# B&R Automation Studio project GAT
Automation Studio 4.10.3.60 SP; technology packages: mapp 5.16.1, mappCockpit 5.16.0, mappControl 5.16.0, mappMotion 5.16.0, mappView 5.16.1

## Configuration 4PPC50_101E_10B

CPU 4PPC50.101E-10B, AutomationRuntime C4.91, Build 4.1.2, Safety 0.0, Vc 

### Task classes (Cpu.sw)
```
Cyclic#1 (cycle 1600 us, tolerance 1600 us):
  MainCtrl <- MainControl.MainCtrl.prg [disabled]
  CrossCutte <- MachineControl.CrossCutter.CrossCutter.prg
  Conveyor <- MachineControl.Conveyor.Conveyor.prg
  AlarmUI <- (binary)
Cyclic#2 (cycle 20000 us, tolerance 20000 us):
  AlarmMgt <- Infrastructure.Alarm.AlarmMgt.prg
Cyclic#4 (cycle 80000 us, tolerance 80000 us):
  AuditMgt <- Infrastructure.Audit.AuditMgt.prg
  ReportMgt <- Infrastructure.Report.ReportMgt.prg
  DataMgt <- Infrastructure.Data.DataMgt.prg
  ProcessCon <- Infrastructure.SysServices.ProcessConfig.prg [disabled]
  PIDControl <- MainControl.PIDControl.prg [disabled]
  RecipeMgt <- Infrastructure.Recipe.RecipeMgt.prg
  IoBrowser <- Infrastructure.SysServices.IoBrowser.prg
  UsbDevLink <- Infrastructure.UsbDevLink.UsbDevLink.prg
Cyclic#5 (cycle 200000 us, tolerance 200000 us):
  SysServs <- Infrastructure.SysServices.SysServs.prg
Cyclic#8 (cycle 8000 us, tolerance 30000000 us):
  UserXMgt <- Infrastructure.UserX.UserXMgt.prg
  UserMgt <- Infrastructure.User.UserMgt.prg [disabled]
DataObjects: McAcpSys
NcDataObjects: McDriveLog
Binaries: arsvcreg, FWRules, McAcpDrv, McAcpSim, mvLoader, McProfGen, McMechSys, TCData, TCLang, udbdef, arcoal, arflatprv, mCoWebSc, OpcUaSrv, arconfig, User, Role, iomap, asfw, ashwac, ashwd, sysconf, TC, Report, Rcp, AlmHistory, Data, Audit, UserXlogin, UsX, Settings, AxCfg, Alarm, CutCamAut, myUnits, FileMgr, CutterAlm, ConvGrp, MachineGrp, Cutter, ConvAlm, CutterGrp, aruser, File, FileMgrRep, FileMgrDat, FileMgrAud, FileUI, CamAutoMa1, User_1, Config, Config_32, AlmCutter, Config_1, Config_2, UserMgr, UserSign, UserLogin, profiler, Config_31, Config_3, CfgUser, Login, Config_23, Config_24, Config_21, Config_20, CamAutoMat, vConfig_0, Config_0, Config_13, Config_5, Config_8, Config_9, Config_11, Config_15, Config_14, Config_12, Config_10, Config_6, Config_7, Config_22, Config_4, Master, Slave, CamID, CamList, ProfGen, vMaster
Libraries: McBase, McAcpAx, McPathGen, McPureVAx, McAxGroup, McAxis, McAcpPar, McProgInt, MpTool, MpAxis, MpBase, MpWebXs, MpAudit, MpRecipe, MpReport, MpFile, MpAlarmX, MpCom, MpBackup, AsArSdm, FileIO, astime, sys_lib, runtime, MpServer, MpData, DataObj, brsystem, CoTrace, AsZip, MpUserX, AsUPS, MTBasics, MTTypes, Gat, AsIO, AsBrStr, AsIOMMan, IoMapMan, ArCfgMan, AsUSB, powerlnk, arssl, arproject, asarlog, asarprof, asmem, asarcfg, asieccon, asstring, asepl, aseth, ashw, arcert, dvframe, standard, mpregmark
```

### Hardware
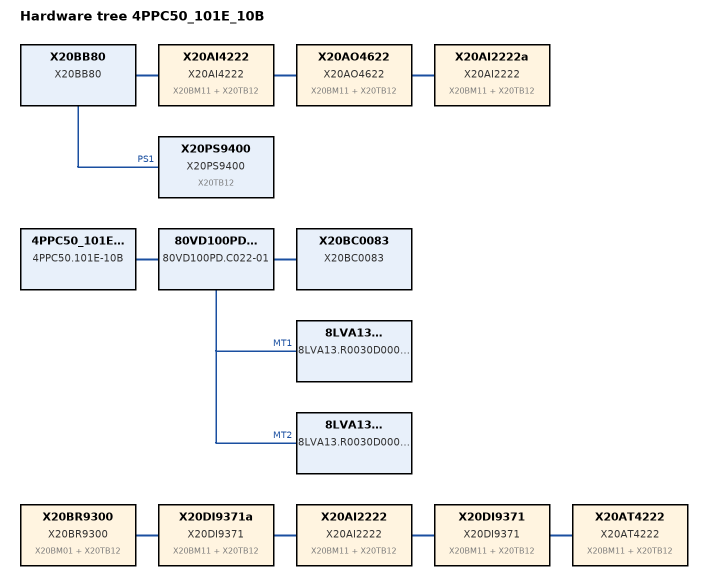
```
4PPC50_101E_10B : 4PPC50.101E-10B v1.1.2.1
  Connector IF1:
    CycleTime = 800
  Connector IF2:
    ActivateDevice = 1
    Mode = Manual
    InternetAddress = 10.86.50.12
    SubnetMask = 255.255.255.0
  Connector IF3:
    AssignedOperatingSystem = ARemb
  Connector IF4:
    AssignedOperatingSystem = GPOS
  ConfigurationID = GAT_10inC50_4PPC50_101E_10B
  UserPartitionSize = 25
  UserRamSize = 16000
  RemMemSize = 48000
  TimerDeviceType = EPLX2X
  TimerDevice = 4PPC50_101E_10B.IF1
  TaskClassIdleTime = 4000
  Cyclic1Duration = 1600
  Cyclic1Tolerance = 1600
  Cyclic1Stack = 16384
  Cyclic2Duration = 20000
  Cyclic2Tolerance = 20000
  Cyclic3Duration = 40000
  Cyclic3Tolerance = 40000
  Cyclic4Duration = 80000
  Cyclic4Tolerance = 80000
  Cyclic4Stack = 16384
  Cyclic5Duration = 200000
  Cyclic5Tolerance = 200000
  Cyclic6Duration = 500000
  Cyclic6Tolerance = 500000
  Cyclic7Duration = 1000000
  Cyclic7Tolerance = 1000000
  Cyclic8Duration = 8000
  Cyclic8Tolerance = 30000000
  FileDevice1
  FileDeviceName1 = mappRecipe
  FileDevicePath1 = F:\GAT\Recipe
  FileDevice2
  FileDeviceName2 = mappAudit
  FileDevicePath2 = F:\GAT\Audit
  FileDevice3
  FileDeviceName3 = mappReport
  FileDevicePath3 = F:\GAT\Report
  FileDevice4
  FileDeviceName4 = mappData
  FileDevicePath4 = F:\GAT\Data
  TimeZone = 295
  EthernetDefaultGateway = 10.86.13.1
  FTPProtocol = 2
  FtpUser1
  FtpUsername1 = BR
  FtpUserPassword1 = GhNaeKiLvl7cP7K0k5JDdXf+fyc8NJfckbGpEUwY4Hg=  // FTP
  FtpUserSalt1 = zT8zXD9V
  FTPAccessRight1 = 0
  FTPdevice1 = ALL
  ActivateOpcUa = 1
  OpcUaActivateAuditEvents = 1
  OpcUa_Security_AdminRole = Administrators
  OpcUaInformationModels_PV_Version = 1
  LXTMode = Manual
  LXTInternetAddress = 10.86.50.13
  LXTSubnetmask = 255.255.255.0
80VD100PD.C022-01 : 80VD100PD.C022-01 v2.5.0.0  [PLK1 -> 4PPC50_101E_10B.IF1 (NodeNumber=1) [Cable Type=PowerlinkCable, Length=10, Version=1.0.0.3]; PLK2 -> X20BC0083.PLK1 (NodeNumber=1) [Cable Type=PowerlinkCable, Length=10, Version=1.0.0.3]; MT2 -> 8LVA13.R0030D000-0a.MT]
  DriveConfiguration/Module:
    McAcoposTypeID = AcoposMicroDConfig
    ActivateACOPOSSimulationOnPLC = 1
  DriveConfiguration/Encoder/EncoderX6A/InterfaceType:
    ResolverPolepairs = 1
  DriveConfiguration/Encoder/EncoderX6B/InterfaceType:
    ResolverPolepairs = 1
  DriveConfiguration/Channel[1]/RealAxis:
    AxisReference = gAxisConveyor
  DriveConfiguration/Channel[1]/RealAxis/MechanicalElements/Gearbox:
    InputIsReadOnly = 0
    Input = 1
    OutputIsReadOnly = 0
    Output = 1
  DriveConfiguration/Channel[1]/RealAxis/MechanicalElements/RotaryToLinearTransformation:
    ReferenceDistanceIsReadOnly = 0
    ReferenceDistance = 1
  DriveConfiguration/Channel[1]/RealAxis/Controller:
    ModeIsReadOnly = 0
    Mode = PositionController
  DriveConfiguration/Channel[1]/RealAxis/Controller/Mode/Position:
    ProportionalGain = 50.0
    IntegrationTime = 0.0
    PredictionTime = 0.0004
    TotalDelayTime = 0.0004
  DriveConfiguration/Channel[1]/RealAxis/Controller/Mode/Speed:
    ProportionalGainIsReadOnly = 0
    ProportionalGain = 2.0
    IntegrationTimeIsReadOnly = 0
    IntegrationTime = 0.0
    FilterTimeIsReadOnly = 0
    FilterTime = 0.0
  DriveConfiguration/Channel[1]/RealAxis/Controller/Mode/LoopFilters:
    LoopFilter1 = NotUsed
    LoopFilter2 = NotUsed
    LoopFilter3 = NotUsed
  DriveConfiguration/Channel[1]/RealAxis/Homing:
    Mode = Direct
  DriveConfiguration/Channel[1]/RealAxis/Homing/Mode:
    Position = 0.0
    ReferencePulse = NotUsed
  DriveConfiguration/Channel[1]/RealAxis/Homing:
    RestorePositionVariable = 
  DriveConfiguration/Channel[1]/RealAxis/StopReaction:
    Quickstop = DecelerationLimit
    DriveError = DecelerationLimit
  DriveConfiguration/Channel[1]/RealAxis/MovementErrorLimits:
    PositionError = 1.0
    VelocityErrorMonitoring = Automatic1
  DriveConfiguration/Channel[1]/RealAxis:
    JerkFilter = NotUsed
  DriveConfiguration/Channel[1]/RealAxis/DigitalInputs/HomingSwitch:
    Source = NotUsed
    Level = High
  DriveConfiguration/Channel[1]/RealAxis/DigitalInputs/PositiveLimitSwitch:
    Source = NotUsed
    Level = High
  DriveConfiguration/Channel[1]/RealAxis/DigitalInputs/NegativeLimitSwitch:
    Source = NotUsed
    Level = High
  DriveConfiguration/Channel[1]/RealAxis/DigitalInputs/Trigger1:
    Source = X2Trigger1
    Level = High
  DriveConfiguration/Channel[1]/RealAxis/DigitalInputs/Trigger2:
    Source = X2Trigger2
    Level = High
  DriveConfiguration/Channel[1]/RealAxis/DigitalInputs/Quickstop:
    Input = Trigger2
  DriveConfiguration/Channel[1]/RealAxis/Simulation:
    SimulationModeOnPLC = SetValueGeneration
    SimulationModeOnACOPOS = NotUsed
  DriveConfiguration/Channel[2]/RealAxis:
    AxisReference = gAxisCrossCutter
  DriveConfiguration/Channel[2]/RealAxis/MechanicalElements/Gearbox:
    InputIsReadOnly = 0
    Input = 1
    OutputIsReadOnly = 0
    Output = 1
  DriveConfiguration/Channel[2]/RealAxis/MechanicalElements/RotaryToLinearTransformation:
    ReferenceDistanceIsReadOnly = 0
    ReferenceDistance = 1
  DriveConfiguration/Channel[2]/RealAxis/Controller:
    ModeIsReadOnly = 0
    Mode = PositionController
  DriveConfiguration/Channel[2]/RealAxis/Controller/Mode/Position:
    ProportionalGain = 50.0
    IntegrationTime = 0.0
    PredictionTime = 0.0004
    TotalDelayTime = 0.0004
  DriveConfiguration/Channel[2]/RealAxis/Controller/Mode/Speed:
    ProportionalGainIsReadOnly = 0
    ProportionalGain = 2.0
    IntegrationTimeIsReadOnly = 0
    IntegrationTime = 0.0
    FilterTimeIsReadOnly = 0
    FilterTime = 0.0
  DriveConfiguration/Channel[2]/RealAxis/Controller/Mode/LoopFilters:
    LoopFilter1 = NotUsed
    LoopFilter2 = NotUsed
    LoopFilter3 = NotUsed
  DriveConfiguration/Channel[2]/RealAxis/Homing:
    Mode = Direct
  DriveConfiguration/Channel[2]/RealAxis/Homing/Mode:
    Position = 0.0
    ReferencePulse = NotUsed
  DriveConfiguration/Channel[2]/RealAxis/Homing:
    RestorePositionVariable = 
  DriveConfiguration/Channel[2]/RealAxis/StopReaction:
    Quickstop = DecelerationLimit
    DriveError = DecelerationLimit
  DriveConfiguration/Channel[2]/RealAxis/MovementErrorLimits:
    PositionError = 1.0
    VelocityErrorMonitoring = Automatic1
  DriveConfiguration/Channel[2]/RealAxis:
    JerkFilter = NotUsed
  DriveConfiguration/Channel[2]/RealAxis/DigitalInputs/HomingSwitch:
    Source = NotUsed
    Level = High
  DriveConfiguration/Channel[2]/RealAxis/DigitalInputs/PositiveLimitSwitch:
    Source = NotUsed
    Level = High
  DriveConfiguration/Channel[2]/RealAxis/DigitalInputs/NegativeLimitSwitch:
    Source = NotUsed
    Level = High
  DriveConfiguration/Channel[2]/RealAxis/DigitalInputs/Trigger1:
    Source = X2Trigger1
    Level = High
  DriveConfiguration/Channel[2]/RealAxis/DigitalInputs/Trigger2:
    Source = X2Trigger2
    Level = High
  DriveConfiguration/Channel[2]/RealAxis/DigitalInputs/Quickstop:
    Input = Trigger2
  DriveConfiguration/Channel[2]/RealAxis/Simulation:
    SimulationModeOnPLC = SetValueGeneration
    SimulationModeOnACOPOS = NotUsed
  DriveConfiguration/Channel[2]/RealAxis/AxisFeatures:
    FeatureRef[1] = CutterCamAutomat
8LVA13.R0030D000-0 : 8LVA13.R0030D000-0 v2.2.0.4  [MT -> 80VD100PD.C022-01.MT1]
  M1/MotorParameters:
    MOTOR_AMB_TEMP_RATED = 40
8LVA13.R0030D000-0a : 8LVA13.R0030D000-0 v2.2.0.4  [MT -> 80VD100PD.C022-01.MT2]
  M1/MotorParameters:
    MOTOR_AMB_TEMP_RATED = 40
X20AI2222 : X20AI2222 v1.1.0.0  [SS1 -> X20TB12b.SS; SL -> X20BM11a.SL1]
  Supervision = off
X20AI2222a : X20AI2222 v1.1.0.0  [SS1 -> X20TB12h.SS; SL -> X20BM11f.SL1]
  Supervision = off
X20AI4222 : X20AI4222 v1.1.0.0  [SS1 -> X20TB12f.SS; SL -> X20BM11d.SL1]
X20AO4622 : X20AO4622 v1.2.0.0  [SS1 -> X20TB12g.SS; SL -> X20BM11e.SL1]
X20AT4222 : X20AT4222 v1.3.0.0  [SS1 -> X20TB12a.SS; SL -> X20BM11.SL1]
  Supervision = off
X20BB80 : X20BB80 v1.0.2.0
X20BC0083 : X20BC0083 v2.11.1.0  [PLK1 -> 80VD100PD.C022-01.PLK2 (NodeNumber=2) [Cable Type=PowerlinkCable, Length=10, Version=1.0.0.3]; SL -> X20BB80.SL1]
X20BM01 : X20BM01 v2.1.0.0
X20BM11 : X20BM11 v1.0.0.1  [X2X1 -> X20BM11b.X2X2]
X20BM11a : X20BM11 v1.0.0.1  [X2X1 -> X20BM11c.X2X2]
X20BM11b : X20BM11 v1.0.0.1  [X2X1 -> X20BM11a.X2X2]
X20BM11c : X20BM11 v1.0.0.1  [X2X1 -> X20BM01.X2X2]
X20BM11d : X20BM11 v1.0.0.1  [X2X1 -> X20BB80.IF1]
X20BM11e : X20BM11 v1.0.0.1  [X2X1 -> X20BM11d.X2X2]
X20BM11f : X20BM11 v1.0.0.1  [X2X1 -> X20BM11e.X2X2]
X20BR9300 : X20BR9300 v1.1.0.0  [SS1 -> X20TB12.SS; SL -> X20BM01.SL1; X2X1 -> 4PPC50_101E_10B.IF5 [Cable Type=X2XCable, Length=10, Version=1.0.0.3]]
  Supervision = off
X20DI9371 : X20DI9371 v1.1.0.0  [SS1 -> X20TB12c.SS; SL -> X20BM11b.SL1]
X20DI9371a : X20DI9371 v1.1.0.0  [SS1 -> X20TB12d.SS; SL -> X20BM11c.SL1]
X20PS9400 : X20PS9400 v1.5.0.0  [SS1 -> X20TB12e.SS; PS -> X20BB80.PS1]
X20TB12 : X20TB12 v1.0.0.0
X20TB12a : X20TB12 v1.0.0.0
X20TB12b : X20TB12 v1.0.0.0
X20TB12c : X20TB12 v1.0.0.0
X20TB12d : X20TB12 v1.0.0.0
X20TB12e : X20TB12 v1.0.0.0
X20TB12f : X20TB12 v1.0.0.0
X20TB12g : X20TB12 v1.0.0.0
X20TB12h : X20TB12 v1.0.0.0
```

### IoMap.iom - 4PPC50_101E_10B/IoMap.iom
```iecst
VAR_CONFIG
	::SysServs:CpuIoMap.SerialNumber_CPU AT %ID."4PPC50_101E_10B".SerialNumber_CPU;
	::SysServs:CpuIoMap.ModuleID_CPU AT %IW."4PPC50_101E_10B".ModuleID_CPU;
	::SysServs:CpuIoMap.HardwareVariant AT %IW."4PPC50_101E_10B".HardwareVariant;
	::SysServs:CpuIoMap.FirmwareVersion AT %IW."4PPC50_101E_10B".FirmwareVersion;
	::SysServs:CpuIoMap.TemperatureCPU AT %IW."4PPC50_101E_10B".TemperatureCPU;
	::SysServs:CpuIoMap.TemperatureENV AT %IW."4PPC50_101E_10B".TemperatureENV;
	::SysServs:CpuIoMap.TerminalTemperatureCPU AT %IW."4PPC50_101E_10B".TerminalTemperatureCPU;
	::SysServs:CpuIoMap.TerminalOK AT %IX."4PPC50_101E_10B".TerminalOk;
	::SysServs:CpuIoMap.TerminalStatus AT %IB."4PPC50_101E_10B".TerminalStatus;
	::SysServs:CpuIoMap.TerminalLoadCPU0 AT %IB."4PPC50_101E_10B".TerminalLoadCPU0;
	::SysServs:CpuIoMap.TerminalLoadCPU1 AT %IB."4PPC50_101E_10B".TerminalLoadCPU1;
	::AlarmMgt:SafetyInputs.SafetyPLC AT %IX."X20DI9371".DigitalInput02;
	::AlarmMgt:SafetyInputs.EmergencyStop[0]  AT %IX."X20DI9371a".DigitalInput06;
END_VAR
```

### AxCfg.axis - 4PPC50_101E_10B/mappMotion/AxCfg.axis
```
Element gAxisConveyor (Type=axis)
  BaseTypeIsReadOnly = 0
  BaseType = Linear
    MeasurementUnit = 5066068
    MeasurementResolutionIsReadOnly = 0
    MeasurementResolution = 0.01
    CountDirectionIsReadOnly = 0
    CountDirection = Standard
  MovementLimitsIsReadOnly = 0
  MovementLimits = Internal
    Position:
      LowerLimitMin = -1.79769313486231E308
      UpperLimitMax = 1.79769313486231E308
      LowerLimit = -1000000000000000000000.0
      UpperLimit = 1000000000000000000000.0
    VelocityIsReadOnly = 0
    Velocity:
      VelocityMax = 3.4E38
      Velocity = 10000
    AccelerationIsReadOnly = 0
    Acceleration:
      AccelerationMax = 3.4E38
      Acceleration = 50000
    DecelerationIsReadOnly = 0
    Deceleration:
      DecelerationMax = 3.4E38
      Deceleration = 50000
  Alarms = MpAlarmX
    mapp.AlarmX.Core.Configuration:
      [0]:
        Message = {$MpMotion/Alarms/System}
      [1]:
        Message = {$MpMotion/Alarms/Initialization}
      [2]:
        Message = {$MpMotion/Alarms/Parameter}
      [3]:
        Message = {$MpMotion/Alarms/Operation}
      [4]:
        Message = {$MpMotion/Alarms/DataAccess}
      [5]:
        Message = {$MpMotion/Alarms/Syntax}
      [9]:
        Message = {$MpMotion/Alarms/Network}
      [10]:
        Message = {$MpMotion/Alarms/Encoder}
        AdditionalInformation1 = Something wrong with the encoder inside the motor
      [11]:
        Message = {$MpMotion/Alarms/Drive}
        AdditionalInformation1 = Acopos Drive Error
      [12]:
        Message = {$MpMotion/Alarms/IO}
      [13]:
        Message = {$MpMotion/Alarms/Supply}
      [14]:
        Message = {$MpMotion/Alarms/Motor}
      [15]:
        Message = {$MpMotion/Alarms/HoldingBrake}
Element gAxisCrossCutter (Type=axis)
  BaseTypeIsReadOnly = 0
  BaseType = RotaryPeriodic
    MeasurementUnitIsReadOnly = 0
    MeasurementUnit = 17476
    MeasurementResolutionIsReadOnly = 0
    MeasurementResolution = 0.01
    CountDirectionIsReadOnly = 0
    CountDirection = Inverse
    PeriodSettings:
      Period = 360
  MovementLimitsIsReadOnly = 0
  MovementLimits = Internal
    Position:
      LowerLimitMin = -1.79769313486231E308
      UpperLimitMax = 1.79769313486231E308
      LowerLimit = -1000.0
      UpperLimit = 1000.0
    VelocityIsReadOnly = 0
    Velocity:
      VelocityMax = 3.4E38
      Velocity = 500000
    AccelerationIsReadOnly = 0
    Acceleration:
      AccelerationMax = 3.4E38
      Acceleration = 5000000
    DecelerationIsReadOnly = 0
    Deceleration:
      DecelerationMax = 3.4E38
      Deceleration = 5000000
  Alarms = MpAlarmX
    mapp.AlarmX.Core.Configuration:
      [0]:
        Message = {$MpMotion/Alarms/System}
      [1]:
        Message = {$MpMotion/Alarms/Initialization}
      [2]:
        Message = {$MpMotion/Alarms/Parameter}
      [3]:
        Message = {$MpMotion/Alarms/Operation}
      [4]:
        Message = {$MpMotion/Alarms/DataAccess}
      [5]:
        Message = {$MpMotion/Alarms/Syntax}
      [9]:
        Message = {$MpMotion/Alarms/Network}
      [10]:
        Message = {$MpMotion/Alarms/Encoder}
      [11]:
        Message = {$MpMotion/Alarms/Drive}
      [12]:
        Message = {$MpMotion/Alarms/IO}
      [13]:
        Message = {$MpMotion/Alarms/Supply}
      [14]:
        Message = {$MpMotion/Alarms/Motor}
      [15]:
        Message = {$MpMotion/Alarms/HoldingBrake}
```

### Alarm.mpalarmxcore - 4PPC50_101E_10B/mappServices/Alarm.mpalarmxcore
```
Element gAlarmXMpLink (Type=mpalarmxcore)
  mapp.AlarmX.Core:
    Mapping:
      [0]:
        Alarm = gAxisMaster*
        [0] = Reaction
          Name = MasterWaitAcknowledge
      [1]:
        Alarm = gAxisSlave*
        [0] = Reaction
          Name = SlaveWaitAcknowledge
    BySeverity:
      [0]:
        Severity = 1
        [0] = Reaction
          Name = StopMovements
      [1]:
        Severity = 10
        [0] = Reaction
      [2]:
        Severity = 20
        [0] = Reaction
  mapp.AlarmX.Core.Configuration:
    [0]:
      Name = FeederSpeedNotSet
      Message = {$AlarmTexts/FeederSpeedNotSet}
      Code = 250
      Severity = 10
    [1]:
      Name = CutterSpeedNotSet
      Message = {$AlarmTexts/CutterSpeedNotSet}
      Code = 251
      Severity = 10
    [2]:
      Name = CutterPositionNotSet
      Message = {$AlarmTexts/CutterPositionNotSet}
      Code = 252
      Severity = 10
    [3]:
      Name = PidOscTuningError
      Message = {$AlarmTexts/PidOscTuningError}
      Behavior = DiscreteValueMonitoring
        Monitoring:
          MonitoredPV = ::PIDControl:MTBasicsOscillationTuning_0.StatusID
          TriggerValues:
            [0] = -1999999999..-1000000000
    [4]:
      Name = PidControlError
      Message = {$AlarmTexts/PidControlError}
      Behavior = DiscreteValueMonitoring
        Monitoring:
          MonitoredPV = ::PIDControl:MTBasicsPID_0.StatusID
          TriggerValues:
            [0] = -1999999999..-1000000000
    [5]:
      Name = PidControlWarning
      Message = {$AlarmTexts/PidControlWarning}
      Behavior = DiscreteValueMonitoring
        Monitoring:
          MonitoredPV = ::PIDControl:MTBasicsPID_0.StatusID
          TriggerValues:
            [0] = -2999999999..-2000000000
    [6]:
      Name = SetCamFailed
      Message = {$AlarmTexts/SetCamFailed}
    [7]:
      Name = EmergencyStop_0
      Message = {$AlarmTexts/EmergencyStop.0}
      Behavior = DiscreteValueMonitoring
        Recording:
          ActiveToInactive = TRUE
        Monitoring:
          MonitoredPV = ::AlarmMgt:SafetyInputs.EmergencyStop[0]
          TriggerValues:
            [0] = 1
    [8]:
      Name = EmergencyStop_1
      Message = {$AlarmTexts/EmergencyStop.1}
      Behavior = DiscreteValueMonitoring
        Recording:
          ActiveToInactive = TRUE
        Monitoring:
          MonitoredPV = ::AlarmMgt:SafetyInputs.EmergencyStop[1]
          TriggerValues:
            [0] = 1
    [9]:
      Name = EmergencyStop_2
      Message = {$AlarmTexts/EmergencyStop.2}
      Behavior = DiscreteValueMonitoring
        Recording:
          ActiveToInactive = TRUE
        Monitoring:
          MonitoredPV = ::AlarmMgt:SafetyInputs.EmergencyStop[2]
          TriggerValues:
            [0] = 1
    [10]:
      Name = SafetyDoor_0
      Message = {$AlarmTexts/SafetyDoor.0}
      Behavior = DiscreteValueMonitoring
        Recording:
          ActiveToInactive = TRUE
        Monitoring:
          MonitoredPV = ::AlarmMgt:SafetyInputs.SafetyDoor[0]
          TriggerValues:
            [0] = 1
    [11]:
      Name = SafetyDoor_1
      Message = {$AlarmTexts/SafetyDoor.1}
      Behavior = DiscreteValueMonitoring
        Recording:
          ActiveToInactive = TRUE
        Monitoring:
          MonitoredPV = ::AlarmMgt:SafetyInputs.SafetyDoor[1]
          TriggerValues:
            [0] = 1
    [12]:
      Name = SafetyDoor_2
      Message = {$AlarmTexts/SafetyDoor.2}
      Behavior = DiscreteValueMonitoring
        Recording:
          ActiveToInactive = TRUE
        Monitoring:
          MonitoredPV = ::AlarmMgt:SafetyInputs.SafetyDoor[2]
          TriggerValues:
            [0] = 1
    [13]:
      Name = SafetyDoor_3
      Message = {$AlarmTexts/SafetyDoor.3}
      Behavior = DiscreteValueMonitoring
        Recording:
          ActiveToInactive = TRUE
        Monitoring:
          MonitoredPV = ::AlarmMgt:SafetyInputs.SafetyDoor[3]
          TriggerValues:
            [0] = 1
    [14]:
      Name = SafetyDoor_4
      Message = {$AlarmTexts/SafetyDoor.4}
      Behavior = DiscreteValueMonitoring
        Recording:
          ActiveToInactive = TRUE
        Monitoring:
          MonitoredPV = ::AlarmMgt:SafetyInputs.SafetyDoor[4]
          TriggerValues:
            [0] = 1
    [15]:
      Name = SafetyDoor_5
      Message = {$AlarmTexts/SafetyDoor.5}
      Behavior = DiscreteValueMonitoring
        Recording:
          ActiveToInactive = TRUE
        Monitoring:
          MonitoredPV = ::AlarmMgt:SafetyInputs.SafetyDoor[5]
          TriggerValues:
            [0] = 1
    [16]:
      Name = SafetyPLC
      Message = {$AlarmTexts/SafetyPLC}
      Behavior = DiscreteValueMonitoring
        Recording:
          ActiveToInactive = TRUE
        Monitoring:
          MonitoredPV = ::AlarmMgt:SafetyInputs.SafetyPLC
          TriggerValues:
            [0] = 1
  mapp.AlarmX.Core.Snippets:
    AutoDetect = 1
    [0]:
      Key = CutterSpeed
      Value:
        PV = ::MainCtrl:AxisControl[1].Status.ActVelocity
    [1]:
      Key = CutterPosition
      Value:
        PV = ::MainCtrl:AxisControl[1].Status.ActPosition
    [2]:
      Key = PidTuningError
      Value:
        PV = ::PIDControl:MTBasicsOscillationTuning_0.StatusID
    [3]:
      Key = PidControlError
      Value:
        PV = ::PIDControl:MTBasicsPID_0.StatusID
  mapp.AlarmX.Core.Categories:
    [0]:
      Name = Information
      SourceProperty:
        Severity = 20
    [1]:
      Name = Warning
      SourceProperty:
        Severity = 10
    [2]:
      Name = Error
      SourceProperty:
        Severity = 1
```

### AlmHistory.mpalarmxhistory - 4PPC50_101E_10B/mappServices/AlmHistory.mpalarmxhistory
```
Element gAlarmXHistoryMpLink (Type=mpalarmxhistory)
  mapp.AlarmX.History:
    Memory:
      MemorySize = 6000
    Auditing = MpAudit
```

### ConvAlm.mpalarmxcore - 4PPC50_101E_10B/mappServices/Conveyor/ConvAlm.mpalarmxcore
```
Element gAlarmXCore_Conveyor (Type=mpalarmxcore)
  mapp.AlarmX.Core:
    BySeverity:
      [0]:
        Severity = 1..9
        [0] = Reaction
          Name = Info
        [1] = Escalate
      [1]:
        Severity = 10..19
        [0] = Reaction
          Name = Warning
        [1] = Escalate
      [2]:
        Severity = 20..29
        [0] = Reaction
          Name = Alarm
        [1] = Escalate
      [3]:
        Severity = 30..39
        [0] = Reaction
          Name = Safety
        [1] = Escalate
  mapp.AlarmX.Core.Configuration:
    [0]:
      Name = ReferenceRequired
      Message = {$IAT/Conveyor/Info/Name} : {$IAT/Conveyor/Alarms/ReferenceRequired}
      Severity = 10
      Behavior = DiscreteValueMonitoring
        Monitoring:
          MonitoredPV = ::Conveyor:AxisControl.Status.ReferenceRequired
          TriggerValues:
            [0] = 1
```

### ConvGrp.mpcomgroup - 4PPC50_101E_10B/mappServices/Conveyor/ConvGrp.mpcomgroup
```
Element gGroupConveyor (Type=mpcomgroup)
  Linking:
    Subnodes:
      0 = gAxisConveyor
      1 = gAlarmXCore_Conveyor
  Alarms = MpAlarmX
```

### CutterAlm.mpalarmxcore - 4PPC50_101E_10B/mappServices/CrossCutter/CutterAlm.mpalarmxcore
```
Element gAlarmXCore_Cutter (Type=mpalarmxcore)
  mapp.AlarmX.Core:
    BySeverity:
      [0]:
        Severity = 1..9
        [0] = Reaction
          Name = Info
        [1] = Escalate
      [1]:
        Severity = 10..19
        [0] = Reaction
          Name = Warning
        [1] = Escalate
      [2]:
        Severity = 20..29
        [0] = Reaction
          Name = Alarm
        [1] = Escalate
      [3]:
        Severity = 30..39
        [0] = Reaction
          Name = Safety
        [1] = Escalate
  mapp.AlarmX.Core.Configuration:
    [0]:
      Name = ReferenceRequired
      Message = {$IAT/CrossCutter/Info/Name} : {$IAT/CrossCutter/Alarms/ReferenceRequired}
      Severity = 10
      Behavior = DiscreteValueMonitoring
        Monitoring:
          MonitoredPV = ::CrossCutte:AxisControl.Status.ReferenceRequired
          TriggerValues:
            [0] = 1
```

### CutterGrp.mpcomgroup - 4PPC50_101E_10B/mappServices/CrossCutter/CutterGrp.mpcomgroup
```
Element gGroupCutter (Type=mpcomgroup)
  Linking:
    Subnodes:
      0 = gAlarmXCore_Cutter
      1 = gAxisCrossCutter
  Alarms = MpAlarmX
```

### Data.mpdatarecorder - 4PPC50_101E_10B/mappServices/Data.mpdatarecorder
```
Element gDataRecorderMpLink (Type=mpdatarecorder)
  DataRecorder:
    MaxFileSize = 10000
    SaveInterval = 2000
    Format = PDF
      Font = 3
      OwnerPassword = 
      AllowCopy = TRUE
      AllowEdit = TRUE
    UnitDefinition = MeasurementSystemBased
      UnitDisplay = 1
  Alarms = MpAlarmX
```

### FileMgr.mpfilemanagerui - 4PPC50_101E_10B/mappServices/FileMgr.mpfilemanagerui
```
Element gDatFileMgrUIMpLink (Type=mpfilemanagerui)
  Alarms = MpAlarmX
Element gRprtFileMgrUIMpLink (Type=mpfilemanagerui)
  Alarms = MpAlarmX
Element gAuditFileMgrUIMpLink (Type=mpfilemanagerui)
  Alarms = MpAlarmX
Element gRecFileMgrUIMpLink (Type=mpfilemanagerui)
  Alarms = MpAlarmX
Element gFileMgrUIMpLink (Type=mpfilemanagerui)
  Alarms = MpAlarmX
```

### MachineGrp.mpcomgroup - 4PPC50_101E_10B/mappServices/MachineGrp.mpcomgroup
```
Element gGroup (Type=mpcomgroup)
  Linking:
    Subnodes:
      0 = gGroupCutter
      1 = gGroupConveyor
      2 = gAlarmXMpLink
  Alarms = MpAlarmX
```

### Rcp.mprecipexml - 4PPC50_101E_10B/mappServices/Rcp.mprecipexml
```
Element gRecipeXmlMpLink (Type=mprecipexml)
  mapp.Recipe.Xml:
    Auditing = MpAudit
  Alarms = MpAlarmX
    mapp.AlarmX.Core.Configuration:
      [0]:
        Message = {$MpRecipeXml/Alarms/SaveFailed}
      [1]:
        Message = {$MpRecipeXml/Alarms/SaveFailedPartial}
      [2]:
        Message = {$MpRecipeXml/Alarms/LoadFailed}
      [3]:
        Message = {$MpRecipeXml/Alarms/LoadFailedPartial}
Element gRecipeXmlPreviewMpLink (Type=mprecipexml)
  Alarms = MpAlarmX
    mapp.AlarmX.Core.Configuration:
      [0]:
        Message = {$MpRecipeXml/Alarms/SaveFailed}
        Severity = 10
      [1]:
        Message = {$MpRecipeXml/Alarms/SaveFailedPartial}
        Severity = 10
      [2]:
        Message = {$MpRecipeXml/Alarms/LoadFailed}
        Severity = 10
      [3]:
        Message = {$MpRecipeXml/Alarms/LoadFailedPartial}
        Severity = 10
```

### Report.mpreportcore - 4PPC50_101E_10B/mappServices/Report.mpreportcore
```
Element gReportMpLink (Type=mpreportcore)
  MpReport:
    Settings:
      ResourceDeviceName = mappReport
      LanguageDependent:
        [0]:
          Language = en
          Font = 1
        [1]:
          Language = zh-CN
    PageLayouts:
      [0]:
        Name = Default
    Styles:
      Text:
        [0]:
          Name = Default
          Size = 12
        [1]:
          Name = Header
          Style = 1
          Size = 20
          Color = FF9900
        [2]:
          Name = Subheader
          Size = 16
          Color = FF9900
      Table:
        [0]:
          Name = Default
          Padding = 10
      Line:
        [0]:
          Name = Default
          Color = FF9900
      Chart:
        PieChart:
          [0]:
            Name = Default
            BorderWidth = 0
        LineChart:
          [0]:
            Name = Default
        BarChart:
          [0]:
            Name = Default
    Tables:
      [0]:
        Name = Information
        TableStyle = Default
        TextStyle = Default
        [0]:
          [0] = TextId
            Source = RecipeName
            Width = 50
          [1] = ValueId
            Value:
              ProcessVariable = ::RecipeMgt:MpRecipeXml_0.Info.LastLoadedRecipe
            Width = 50
        [1]:
          [0] = TextId
            Source = Index
            Width = 50
          [1] = TextId
            Source = Length [mm]
            Width = 50
          [2] = TextId
            Source = Number
            Width = 50
        [2]:
          [0] = TextId
            Source = 1
            Width = 50
          [1] = ValueId
            Value:
              ProcessVariable = ::MainCtrl:MainCtrl.Para.ProductLength[0]
            Width = 50
          [2] = ValueId
            Value:
              ProcessVariable = ::MainCtrl:MainCtrl.Para.ProductNumber[0]
            Width = 50
        [3]:
          [0] = TextId
            Source = 2
            Width = 50
          [1] = ValueId
            Value:
              ProcessVariable = ::MainCtrl:MainCtrl.Para.ProductLength[1]
            Width = 50
          [2] = ValueId
            Value:
              ProcessVariable = ::MainCtrl:MainCtrl.Para.ProductNumber[1]
            Width = 50
        [4]:
          [0] = TextId
            Source = 3
            Width = 50
          [1] = ValueId
            Value:
              ProcessVariable = ::MainCtrl:MainCtrl.Para.ProductLength[2]
            Width = 50
          [2] = ValueId
            Value:
              ProcessVariable = ::MainCtrl:MainCtrl.Para.ProductNumber[2]
            Width = 50
        [5]:
          [0] = TextId
            Source = 4
            Width = 50
          [1] = ValueId
            Value:
              ProcessVariable = ::MainCtrl:MainCtrl.Para.ProductLength[3]
            Width = 50
          [2] = ValueId
            Value:
              ProcessVariable = ::MainCtrl:MainCtrl.Para.ProductNumber[3]
            Width = 50
        [6]:
          [0] = TextId
            Source = 5
            Width = 50
          [1] = ValueId
            Value:
              ProcessVariable = ::MainCtrl:MainCtrl.Para.ProductLength[4]
            Width = 50
          [2] = ValueId
            Value:
              ProcessVariable = ::MainCtrl:MainCtrl.Para.ProductNumber[4]
            Width = 50
    Contents:
      [0]:
        Name = ContentHeader
        [0]:
          Text = {Header}
        [1] = DateTime
        [2] = Line
          LineStyle = Default
      [1]:
        Name = ContentTable
        [0] = Table
          Table = Information
          HorizontalAlign = 1
      [2]:
        Name = Header
        [0]:
          Text = Report of the Cross Cutter Machine
          HorizontalAlign = 1
          TextStyle = Header
      [3]:
        Name = EmptyLine
        [0] = EmptyLine
      [4]:
        Name = Underline
        [0] = Line
          LineStyle = Default
      [5]:
        Name = Date
        [0] = DateTime
          TextStyle = Default
    Reports:
      [0]:
        Name = Report
        PageLayout = Default
        Header = Header
        [0]:
          [0]:
            Content = Underline
        [1]:
          [0]:
            Content = EmptyLine
        [2]:
          Heading:
            Text = Time
            TextStyle = Subheader
          [0]:
            Content = Date
        [3]:
          [0]:
            Content = EmptyLine
        [4]:
          [0]:
            Content = EmptyLine
        [5]:
          Heading:
            Text = Data
            TextStyle = Subheader
          [0]:
            Content = ContentTable
  Alarms = MpAlarmX
```

### UsX.mpuserx - 4PPC50_101E_10B/mappServices/UserX/UsX.mpuserx
```
Element UserMgmtX (Type=mpuserx)
  Mgr:
    PasswordLength = 1
    LoginAttempts = 5
  ServerSettings:
    Server:
      AdditionalUserData:
        [0] = mail
        [1] = telephoneNumber
  Users:
    DefUser#1:
      id = Admin
      name = Admin
    DefUser#2:
      id = Anonymous
      name = Anonymous
    DefUser#3:
      id = Operator
      name = Operator
    DefUser#4:
      id = Service_Tech
      name = Service_Tech
  Groups:
    DefGroup#1:
      id = Administrators
      level = 100
      admin = TRUE
      rights:
        [0] = FullAccess
        [1] = ViewOnly
        [2] = StartOnly
    DefGroup#2:
      id = Everyone
      level = 3
      rights:
        [0] = ViewOnly
    DefGroup#3:
      id = Operators
      level = 30
      rights:
        [0] = StartOnly
    DefGroup#4:
      id = Service
      level = 50
      rights:
        [0] = StartOnly
        [1] = ViewOnly
    DefGroup#5:
      id = Everyone
      level = 3
      rights:
        [0] = ViewOnly
```

### UserXlogin.mpuserxlogin - 4PPC50_101E_10B/mappServices/UserX/UserXlogin.mpuserxlogin
```
Element gUserXLoginMpLink (Type=mpuserxlogin)
  Alarms = MpAlarmX
```

## Configuration PPC2200

CPU 5PPC2200.AL14-000, AutomationRuntime D4.91, Build 4.1.2, Safety 0.0, Vc V4.72.3

### Task classes (Cpu.sw)
```
Cyclic#1 (cycle 1600 us, tolerance 1600 us):
  MainCtrl <- MainControl.MainCtrl.prg [disabled]
  AxisContro <- Infrastructure.AxisTemplate.AxisControl.prg [disabled]
  AppAxis_1 <- MachineControl.AppAxis_1.AppAxis_1.prg
  CrossCutte <- MachineControl.CrossCutter.CrossCutter.prg [disabled]
  AlarmX1 <- (binary)
Cyclic#2 (cycle 3200 us, tolerance 3200 us):
  PIDControl <- MainControl.PIDControl.prg [disabled]
Cyclic#5 (cycle 25600 us, tolerance 25600 us):
  UserMgt <- Infrastructure.User.UserMgt.prg [disabled]
  ProcessCon <- Infrastructure.SysServices.ProcessConfig.prg [disabled]
  AlarmMgr <- Infrastructure.AlarmX.AlarmMgr.prg
  FileMgr <- Infrastructure.File.FileMgr.prg
  ReportMgr <- Infrastructure.Report.ReportMgr.prg
  AuditMgr <- Infrastructure.Audit.AuditMgr.prg
  UserXMgr <- Infrastructure.UserX.UserXMgr.prg
  DataMgr <- Infrastructure.Data.DataMgr.prg
  RecipeMgr <- Infrastructure.Recipe.RecipeMgr.prg
  UsbMgr <- Infrastructure.Usb.UsbMgr.prg
  BackupMgr <- Infrastructure.Backup.BackupMgr.prg
Cyclic#8 (cycle 9600 us):
  IoBrowser <- Infrastructure.SysServices.IoBrowser.prg
  SysServs <- Infrastructure.SysServices.SysServs.prg
DataObjects: McAcpSys
NcDataObjects: McDriveLog
Binaries: TCData, OpcUaSrv, McAcpSim, mCoWebSc, McProfGen, udbdef, TCLang, McAcpDrv, mvLoader, arsvcreg, arflatprv, FWRules, arcoal, Report, Audit, Data, sysconf, CutterAlm, asfw, UserXlogin, MachineGrp, Role, User, Settings, ashwd, ashwac, CutVirt, iomap, arconfig, CutAxis, CutCamAut, myUnits, CutterGrp, TC, BackupFile, Config, RecipeXML, AlarmXHist, RecipeCSV, VAppAxis1, Axis1Alm, Axis1Grp, AppAxis1, RecipeFile, DataFile, ReportFile, AuditFile, Backup, UserX, AlarmX, AuditCfg, FileCfg, BackupCfg, AlarmXCfg, ReportCfg, UserXCfg, DataCfg, Recipe, McMechSys, ConvVirt, ConvAxis, ConvGrp, ConvAlm, Cutter, AlmHistory, Rcp, Alarm, UsX
Libraries: operator, runtime, astime, AsIecCon, brsystem, sys_lib, AsArSdm, FileIO, standard, AsBrStr, asstring, AsBrWStr, ArUser, AsMem, AsARCfg, MTTypes, AsZip, DataObj, AsUPS, AsIO, AsIOMMan, Gat, IoMapMan, ArCfgMan, MTBasics, AsUSB, CoTrace, MpFile, MpData, MpBase, MpAxis, MpWebXs, MpAudit, MpRecipe, MpUserX, MpReport, MpAlarmX, MpCom, MpBackup, McAxis, McBase, McAcpAx, McPureVAx, McAcpPar, MpServer, MpRegMark, dvframe, AsIODiag, aseth, arssl, asepl, powerlnk, ashw, arproject, arcert, LoggingLib, snprintf, asarlog, asarprof
```

### Hardware
```
5AP1130.185C-000 : 5AP1130.185C-000 v2.0.0.0
5PPC2200_AL14_000 : 5PPC2200.AL14-000 v2.0.1.0  [SY -> 5AP1130.185C-000.SY1]
  Connector IF3:
    AssignedOperatingSystem = ARemb
    ActivateDevice = 1
    ActivateSnmp = 1
  Connector IF4:
    AssignedOperatingSystem = GPOS
  Connector IF7:
    OperatingSystem = ARemb
    ActivateDevice = 1
  Connector IF5:
    AssignedOperatingSystem = ARemb
  Connector IF6:
    AssignedOperatingSystem = GPOS
  ConfigurationID = mappFW_PPC2200
  UserPartitionSize = 128
  Simulation = 1
  SystemTick = 1600
  TaskClassIdleTime = 1600
  Cyclic1Duration = 1600
  Cyclic1Tolerance = 1600
  Cyclic2Duration = 3200
  Cyclic2Tolerance = 3200
  Cyclic3Duration = 6400
  Cyclic3Tolerance = 6400
  Cyclic4Duration = 12800
  Cyclic4Tolerance = 12800
  Cyclic5Duration = 25600
  Cyclic5Tolerance = 25600
  Cyclic6Duration = 51200
  Cyclic6Tolerance = 51200
  Cyclic7Duration = 102400
  Cyclic7Tolerance = 102400
  Cyclic8Duration = 9600
  FileDevice1
  FileDeviceName1 = userPartition
  FileDevicePath1 = F:\
  FileDevice2
  FileDeviceName2 = mappRecipeFiles
  FileDevicePath2 = F:\Recipe
  FileDevice3
  FileDeviceName3 = mappAuditFiles
  FileDevicePath3 = F:\Audit
  FileDevice4
  FileDeviceName4 = mappReportFiles
  FileDevicePath4 = F:\Report
  FileDevice5
  FileDeviceName5 = mappDataFiles
  FileDevicePath5 = F:\Data
  FileDevice6
  FileDeviceName6 = mappBackupFiles
  FileDevicePath6 = F:\Backup
  FileDevice7
  FileDeviceName7 = mappAlarmXFiles
  FileDevicePath7 = F:\AlarmX
  FileDevice8
  FileDeviceName8 = mappUserXFiles
  FileDevicePath8 = F:\UserX
  TimeZone = 65
  ActivateDaylightSavingTime = 1
  FtpUser1
  FtpUsername1 = user
  FtpUserPassword1 = sHpIbnZIAriJzdWitYyNPul7Ws1MiS3ggYkn5Z1jgCk=
  FtpUserSalt1 = 13A/KPuX
  FTPAccessRight1 = 0
  FTPdevice1 = ALL
  ActivateOpcUa = 1
  OpcUaInformationModels_PV_Version = 1
  ActivateHypervisor = 1
```

### AlarmMgr.uad.bak - 5PPC2200_AL14_000/Connectivity/OpcUA/AlarmMgr.uad.bak
```
OpcUaSource (FileVersion=7, ArVersion=D4.91)
  Aliases:
    ACLAliases:
      ACL (Id=1)
        ACE (RoleName=Service, Access=0x015F)
        ACE (RoleName=Administrators, Access=0x017F)
        ACE (RoleName=Operators, Access=0x015F)
        ACE (RoleName=Everyone, Access=0x015F)
      ACL (Id=3)
        ACE (RoleName=Service, Access=0x01FF)
        ACE (RoleName=Administrators, Access=0x01FF)
        ACE (RoleName=Operators, Access=0x01FF)
        ACE (RoleName=Everyone, Access=0x017F)
    EURangeViolationAliases
    EURangesAliases
    EngineeringUnitAliases
  DefaultView (AclId=3)
    Module <Default>:
      Task AlarmMgr:
        Variable MpAlarmXCore_0:
          Variable ActiveAlarms
          Variable PendingAlarms
          Variable ErrorReset
          Variable Error
        Variable MpAlarmXHistory_0:
          Variable ErrorReset
          Variable Error
        Variable MpAlarmXHistoryUI_0:
          Variable ErrorReset
          Variable Error
        Variable MpAlarmXListUI_0:
          Variable ErrorReset
          Variable Error
        Variable InstanceID
        Variable MpAlarmXListUIConnect:
          Variable Details:
            Variable Backtrace:
              Variable RecordID (EnableArrayElements=True)
              Variable LogbookName (EnableArrayElements=True)
              Variable EventID (EnableArrayElements=True)
              Variable Description (EnableArrayElements=True)
        Variable HmiAlarmX (AutomaticEnable=True)
          Variable Status:
            Variable TableConfig (EnableArrayElements=True)
        Variable QueryActiveAlarms
        Variable AlarmQuery:
          Variable Alarms (EnableArrayElements=True)
        Variable AlarmQueryHMI (AutomaticEnable=True)
          Variable Active (EnableArrayElements=True)
          Variable Acknowledged (EnableArrayElements=True)
          Variable Scope (EnableArrayElements=True)
          Variable Name (EnableArrayElements=True)
          Variable Message (EnableArrayElements=True)
          Variable AdditionalInfo (EnableArrayElements=True)
          Variable Code (EnableArrayElements=True)
          Variable Severity (EnableArrayElements=True)
          Variable TimeStamp (EnableArrayElements=True)
```

### AlarmMgt.uad.bak - 5PPC2200_AL14_000/Connectivity/OpcUA/AlarmMgt.uad.bak
```
OpcUaSource (FileVersion=7, ArVersion=D4.91)
  Aliases:
    ACLAliases:
      ACL (Id=1)
        ACE (RoleName=Service, Access=0x015F)
        ACE (RoleName=Administrators, Access=0x017F)
        ACE (RoleName=Operators, Access=0x015F)
        ACE (RoleName=Everyone, Access=0x015F)
      ACL (Id=3)
        ACE (RoleName=Service, Access=0x01FF)
        ACE (RoleName=Administrators, Access=0x01FF)
        ACE (RoleName=Operators, Access=0x01FF)
        ACE (RoleName=Everyone, Access=0x017F)
    EURangeViolationAliases
    EURangesAliases
    EngineeringUnitAliases
  DefaultView (AclId=3)
    Module <Default>:
      Task AlarmMgt:
        Variable MpAlarmXCore_0:
          Variable ActiveAlarms
          Variable PendingAlarms
          Variable ErrorReset
          Variable Error
        Variable MpAlarmXHistory_0:
          Variable ErrorReset
          Variable Error
        Variable MpAlarmXHistoryUI_0:
          Variable ErrorReset
          Variable Error
        Variable MpAlarmXListUI_0:
          Variable ErrorReset
          Variable Error
        Variable InstanceID
        Variable MpAlarmXListUIConnect:
          Variable Details:
            Variable Backtrace:
              Variable RecordID (EnableArrayElements=True)
              Variable LogbookName (EnableArrayElements=True)
              Variable EventID (EnableArrayElements=True)
              Variable Description (EnableArrayElements=True)
        Variable HmiAlarmX (AutomaticEnable=True)
          Variable Status:
            Variable TableConfig (EnableArrayElements=True)
        Variable QueryActiveAlarms
        Variable AlarmQuery:
          Variable Alarms (EnableArrayElements=True)
        Variable AlarmQueryHMI (AutomaticEnable=True)
          Variable Active (EnableArrayElements=True)
          Variable Acknowledged (EnableArrayElements=True)
          Variable Scope (EnableArrayElements=True)
          Variable Name (EnableArrayElements=True)
          Variable Message (EnableArrayElements=True)
          Variable AdditionalInfo (EnableArrayElements=True)
          Variable Code (EnableArrayElements=True)
          Variable Severity (EnableArrayElements=True)
          Variable TimeStamp (EnableArrayElements=True)
```

### AlarmX2.uad.bak - 5PPC2200_AL14_000/Connectivity/OpcUA/AlarmX2.uad.bak
```
OpcUaSource (FileVersion=7, ArVersion=D4.91)
  Aliases:
    ACLAliases:
      ACL (Id=1)
        ACE (RoleName=Service, Access=0x015F)
        ACE (RoleName=Administrators, Access=0x017F)
        ACE (RoleName=Operators, Access=0x015F)
        ACE (RoleName=Everyone, Access=0x015F)
      ACL (Id=3)
        ACE (RoleName=Service, Access=0x01FF)
        ACE (RoleName=Administrators, Access=0x01FF)
        ACE (RoleName=Operators, Access=0x01FF)
        ACE (RoleName=Everyone, Access=0x017F)
    EURangeViolationAliases
    EURangesAliases
    EngineeringUnitAliases
  DefaultView (AclId=3)
    Module <Default>:
      Task AlarmX:
        Variable MpAlarmXCore_0:
          Variable ActiveAlarms
          Variable PendingAlarms
          Variable ErrorReset
          Variable Error
        Variable MpAlarmXHistory_0:
          Variable ErrorReset
          Variable Error
        Variable MpAlarmXHistoryUI_0:
          Variable ErrorReset
          Variable Error
        Variable MpAlarmXListUI_0:
          Variable ErrorReset
          Variable Error
        Variable InstanceID
        Variable MpAlarmXListUIConnect:
          Variable Details:
            Variable Backtrace:
              Variable RecordID (EnableArrayElements=True)
              Variable LogbookName (EnableArrayElements=True)
              Variable EventID (EnableArrayElements=True)
              Variable Description (EnableArrayElements=True)
        Variable HmiAlarmX (AutomaticEnable=True)
          Variable Status:
            Variable TableConfig (EnableArrayElements=True)
        Variable QueryActiveAlarms
        Variable AlarmQuery:
          Variable Alarms (EnableArrayElements=True)
        Variable AlarmQueryHMI (AutomaticEnable=True)
          Variable Active (EnableArrayElements=True)
          Variable Acknowledged (EnableArrayElements=True)
          Variable Scope (EnableArrayElements=True)
          Variable Name (EnableArrayElements=True)
          Variable Message (EnableArrayElements=True)
          Variable AdditionalInfo (EnableArrayElements=True)
          Variable Code (EnableArrayElements=True)
          Variable Severity (EnableArrayElements=True)
          Variable TimeStamp (EnableArrayElements=True)
```

### FileMgt.uad.bak - 5PPC2200_AL14_000/Connectivity/OpcUA/FileMgt.uad.bak
```
OpcUaSource (FileVersion=7, ArVersion=D4.91)
  Aliases:
    ACLAliases
    EURangeViolationAliases
    EURangesAliases
    EngineeringUnitAliases
  DefaultView:
    Module <Default>:
      Task FileMgt:
        Variable HmiFile (AutomaticEnable=True)
          Variable Status:
            Variable TableConfig (EnableArrayElements=True)
        Variable MpFileManagerUIConnect (AutomaticEnable=True)
          Variable DeviceList:
            Variable DeviceNames (EnableArrayElements=True)
          Variable File:
            Variable List:
              Variable Items (EnableArrayElements=True)
```

### OpcUaMap.uad.bak - 5PPC2200_AL14_000/Connectivity/OpcUA/OpcUaMap.uad.bak
```
OpcUaSource (FileVersion=7, ArVersion=D4.91)
  Aliases:
    ACLAliases:
      ACL (Id=1)
        ACE (RoleName=Service, Access=0x015F)
        ACE (RoleName=Administrators, Access=0x017F)
        ACE (RoleName=Operators, Access=0x015F)
        ACE (RoleName=Everyone, Access=0x015F)
      ACL (Id=3)
        ACE (RoleName=Service, Access=0x01FF)
        ACE (RoleName=Administrators, Access=0x01FF)
        ACE (RoleName=Operators, Access=0x01FF)
        ACE (RoleName=Everyone, Access=0x017F)
    EURangeViolationAliases
    EURangesAliases:
      EURanges (Id=10)
        EURange:
          Low = 1 (ValueProvider=Const)
          High (ValueProvider=Const)
      EURanges (Id=11)
        EURange:
          Low = 0 (ValueProvider=Const)
          High = 360 (ValueProvider=Const)
      EURanges (Id=12)
        EURange:
          Low = 0 (ValueProvider=Const)
          High (ValueProvider=Const)
      EURanges (Id=14)
        EURange:
          Low = ::MainCtrl:MainCtrl.FixParameter.MinProductLength (ValueProvider=PV)
          High = ::MainCtrl:MainCtrl.FixParameter.MaxProductLength (ValueProvider=PV)
      EURanges (Id=15)
        EURange:
          Low = -100 (ValueProvider=Const)
          High = ::PIDControl:PidControlParameters.MaxOut (ValueProvider=PV)
      EURanges (Id=16)
        EURange:
          Low = ::PIDControl:PidControlParameters.MinOut (ValueProvider=PV)
          High = 100 (ValueProvider=Const)
      EURanges (Id=17)
        EURange:
          Low (ValueProvider=Const)
          High = 32767 (ValueProvider=Const)
    EngineeringUnitAliases:
      EngineeringUnit millimetre (Id=1, UnitId=5066068, NameSpaceUri=http://www.opcfoundation.org/UA/units/un/cefact, Symbol=mm)
      EngineeringUnit Index (Id=2, UnitId=4801624, NameSpaceUri=http://www.br-automation.com/units, Symbol=IDX)
      EngineeringUnit degree [unit of angle] (Id=3, UnitId=17476, NameSpaceUri=http://www.opcfoundation.org/UA/units/un/cefact, Symbol=°)
      EngineeringUnit newton metre (Id=4, UnitId=20053, NameSpaceUri=http://www.opcfoundation.org/UA/units/un/cefact, Symbol=N·m)
      EngineeringUnit millimetre per second (Id=8, UnitId=4403510, NameSpaceUri=http://www.opcfoundation.org/UA/units/un/cefact, Symbol=mm/s)
      EngineeringUnit millimetre per second squared (Id=9, UnitId=5059633, NameSpaceUri=http://www.opcfoundation.org/UA/units/un/cefact, Symbol=mm/s²)
      EngineeringUnit degree per second (Id=10, UnitId=4536630, NameSpaceUri=http://www.opcfoundation.org/UA/units/un/cefact, Symbol=°/s)
      EngineeringUnit degree [unit of angle] per second squared (Id=11, UnitId=5059637, NameSpaceUri=http://www.opcfoundation.org/UA/units/un/cefact, Symbol=°/s²)
      EngineeringUnit second [unit of time] (Id=12, UnitId=5457219, NameSpaceUri=http://www.opcfoundation.org/UA/units/un/cefact, Symbol=s)
      EngineeringUnit deci degree (Id=13, UnitId=4474180, NameSpaceUri=http://www.br-automation.com/units, Symbol=°C/10)
      EngineeringUnit one (Id=14, UnitId=4404786, NameSpaceUri=http://www.opcfoundation.org/UA/units/un/cefact, Symbol=1)
  DefaultView (AclId=3)
    Module <Default>:
      GlobalVariables Global Variables:
        Variable gUSBAvailable (EnableArrayElements=True)
      Task MainCtrl:
        Variable CopyPreviewParameters
        Variable MainCtrl:
          Variable Parameter (AutomaticEnable=True)
            Variable ProductNumber (EnableArrayElements=True)
              Variable ProductNumber[0] (AuditEvents=True)
              Variable ProductNumber[1] (AuditEvents=True)
              Variable ProductNumber[2] (AuditEvents=True)
              Variable ProductNumber[3] (AuditEvents=True)
              Variable ProductNumber[4] (AuditEvents=True)
            Variable ProductLength (EnableArrayElements=True)
              Variable ProductLength[0] (AuditEvents=True, EURangesId=14, EngineeringUnitId=1)
              Variable ProductLength[1] (AuditEvents=True, EURangesId=14, EngineeringUnitId=1)
              Variable ProductLength[2] (AuditEvents=True, EURangesId=14, EngineeringUnitId=1)
              Variable ProductLength[3] (AuditEvents=True, EURangesId=14, EngineeringUnitId=1)
              Variable ProductLength[4] (AuditEvents=True, EURangesId=14, EngineeringUnitId=1)
            Variable AxPar (EnableArrayElements=True)
              Variable AxPar[1]:
                Variable Position (EngineeringUnitId=3)
                Variable Distance (EngineeringUnitId=3)
                Variable Velocity (EngineeringUnitId=10)
                Variable Acceleration (EngineeringUnitId=11)
                Variable Deceleration (EngineeringUnitId=11)
                Variable Stop:
                  Variable Deceleration (EngineeringUnitId=11)
                Variable LimitLoad:
                  Variable Load (EngineeringUnitId=4)
              Variable AxPar[0]:
                Variable Position (EngineeringUnitId=1)
                Variable Distance (EngineeringUnitId=1)
                Variable Velocity (EngineeringUnitId=8)
                Variable Acceleration (EngineeringUnitId=9)
                Variable Deceleration (EngineeringUnitId=9)
                Variable Stop:
                  Variable Deceleration (EngineeringUnitId=9)
                Variable LimitLoad:
                  Variable Load (EngineeringUnitId=4)
          Variable Command:
            Variable AutoModeOn
            Variable RunFeeder
            Variable RunCutter
          Variable Status (AutomaticEnable=True)
            Variable CurrentBatch (EngineeringUnitId=2)
            Variable CurrentBatchLength (EngineeringUnitId=1)
          Variable FixParameter (AutomaticEnable=True)
            Variable SyncAngle (AuditEvents=True, EURangesId=11, EngineeringUnitId=3)
            Variable NrOfKnives (AuditEvents=True, EURangesId=10)
            Variable MaxProductLength (AuditEvents=True, EURangesId=12, EngineeringUnitId=1)
            Variable CutDiameter (AuditEvents=True, EURangesId=12, EngineeringUnitId=1)
            Variable MinProductLength (AuditEvents=True, EURangesId=12, EngineeringUnitId=1)
          Variable Intern:
            Variable ProductNumber (EnableArrayElements=True)
            Variable ProductLength (EnableArrayElements=True)
              Variable ProductLength[0] (EngineeringUnitId=1)
              Variable ProductLength[1] (EngineeringUnitId=1)
              Variable ProductLength[2] (EngineeringUnitId=1)
              Variable ProductLength[3] (EngineeringUnitId=1)
              Variable ProductLength[4] (EngineeringUnitId=1)
        Variable PreviewParameters (AutomaticEnable=True)
          Variable ProductNumber (EnableArrayElements=True)
          Variable ProductLength (EnableArrayElements=True)
            Variable ProductLength[0] (EngineeringUnitId=1)
            Variable ProductLength[1] (EngineeringUnitId=1)
            Variable ProductLength[2] (EngineeringUnitId=1)
            Variable ProductLength[3] (EngineeringUnitId=1)
            Variable ProductLength[4] (EngineeringUnitId=1)
          Variable AxPar (EnableArrayElements=True)
            Variable AxPar[0]:
              Variable Position (EngineeringUnitId=1)
              Variable Distance (EngineeringUnitId=1)
              Variable Velocity (EngineeringUnitId=8)
              Variable Acceleration (EngineeringUnitId=9)
              Variable Deceleration (EngineeringUnitId=9)
              Variable Stop:
                Variable Deceleration (EngineeringUnitId=9)
              Variable LimitLoad:
                Variable Load (EngineeringUnitId=4)
            Variable AxPar[1]:
              Variable Position (EngineeringUnitId=3)
              Variable Distance (EngineeringUnitId=3)
              Variable Velocity (EngineeringUnitId=10)
              Variable Acceleration (EngineeringUnitId=11)
              Variable Deceleration (EngineeringUnitId=11)
              Variable Stop:
                Variable Deceleration (EngineeringUnitId=11)
              Variable LimitLoad:
                Variable Load (EngineeringUnitId=4)
        Variable AxisControl (EnableArrayElements=True)
          Variable AxisControl[0]:
            Variable Parameter:
              Variable AxPar:
                Variable Position (EngineeringUnitId=1)
                Variable Distance (EngineeringUnitId=1)
                Variable Velocity (EURangesId=12, EngineeringUnitId=8)
                Variable Acceleration (EngineeringUnitId=9)
                Variable Deceleration (EngineeringUnitId=9)
                Variable Homing:
                  Variable Position (EngineeringUnitId=1)
                Variable Jog:
                  Variable Velocity (EngineeringUnitId=8)
                  Variable Acceleration (EngineeringUnitId=9)
                  Variable Deceleration (EngineeringUnitId=9)
                  Variable LimitPosition:
                    Variable FirstPosition (EngineeringUnitId=1)
                    Variable LastPosition (EngineeringUnitId=1)
                Variable Stop:
                  Variable Deceleration (EngineeringUnitId=9)
                Variable LimitLoad:
                  Variable Load (EngineeringUnitId=4)
            Variable Status:
              Variable ActPosition (Historizing=True, HistoryBufferSize=2000, HistorySamplingInterval=Timer3, EngineeringUnitId=1)
              Variable ActVelocity (EngineeringUnitId=8)
              Variable ActTorque (EngineeringUnitId=4)
          Variable AxisControl[1]:
            Variable Parameter:
              Variable AxPar:
                Variable Velocity (EURangesId=12, EngineeringUnitId=10)
                Variable Position (EngineeringUnitId=3)
                Variable Distance (EngineeringUnitId=3)
                Variable Acceleration (EngineeringUnitId=11)
                Variable Deceleration (EngineeringUnitId=11)
                Variable Homing:
                  Variable Position (EngineeringUnitId=3)
                Variable Jog:
                  Variable Velocity (EngineeringUnitId=10)
                  Variable Acceleration (EngineeringUnitId=11)
                  Variable Deceleration (EngineeringUnitId=11)
                  Variable LimitPosition:
                    Variable FirstPosition (EngineeringUnitId=3)
                    Variable LastPosition (EngineeringUnitId=3)
                Variable Stop:
                  Variable Deceleration (EngineeringUnitId=11)
                Variable LimitLoad:
                  Variable Load (EngineeringUnitId=4)
            Variable Status:
              Variable ActPosition (Historizing=True, HistoryBufferSize=2000, HistorySamplingInterval=Timer3, EURangesId=11, EngineeringUnitId=3)
              Variable ActVelocity (EngineeringUnitId=10)
              Variable ActTorque (EngineeringUnitId=4)
        Variable MC_BR_CamAutomatCommand_0:
          Variable Ready
          Variable Running
          Variable Error
        Variable MpAxisBasic_x (EnableArrayElements=True)
          Variable MpAxisBasic_x[0]:
            Variable Velocity (EngineeringUnitId=8)
        Variable ResetEditValues
      Task AuditMgt:
        Variable DisplayFileName
        Variable StrSelectedFile
        Variable DisplayFileNameIndex
        Variable MpAuditTrail_0:
          Variable Export
          Variable Error
          Variable ErrorReset
        Variable MpFileManagerUIConnect:
          Variable File:
            Variable Refresh
        Variable TableConfig
      Task ReportMgt:
        Variable DeleteReport
        Variable EnableDelete
        Variable EnableGenerate
        Variable StartGenerate
        Variable SetLanguage
        Variable StrSelectedFile
        Variable DisplayFileNameIndex
        Variable DisplayFileName
        Variable MpReportCore_0:
          Variable ErrorReset
          Variable Error
        Variable TableConfig
      Task DataMgt:
        Variable DisplayFileName
        Variable StrSelectedFile
        Variable DisplayFileNameIndex
        Variable MpDataRecorder_0:
          Variable Record
          Variable ErrorReset
          Variable Error
        Variable MpFileManagerUIConnect:
          Variable File:
            Variable Refresh
        Variable TableConfig
        Variable MpFileManagerUI_0:
          Variable ErrorReset
          Variable Error
      Task UserMgt:
        Variable CreateNewUser
        Variable DataProvider
        Variable idx
        Variable idy
        Variable PropertyName
        Variable ROLE_LISTTYPE
        Variable RoleCounter
        Variable NewUserConfirmPassword
        Variable NewUserName
        Variable NewUserPassword
        Variable tmpUser
        Variable tmpUserIdx
        Variable tmpUserNew
        Variable tmpUserOld
        Variable USER_LISTTYPE
        Variable UserCounter
        Variable UserCounterTotal
        Variable UserManagementState
        Variable USERROLE_LISTTYPE
        Variable Password
        Variable UserName
        Variable ArUserAssignRole_0:
          Variable UserName
          Variable RoleName
        Variable ArUserCreate_0:
          Variable UserName
        Variable ArUserDelete_0:
          Variable UserName
        Variable ArUserDestroyList_0
        Variable ArUserGetFirst_0:
          Variable List
        Variable ArUserGetNext_0:
          Variable List
        Variable ArUserGetProperty_0:
          Variable Execute
          Variable ElementType
          Variable ElementName
          Variable PropertyName
          Variable PropertyValue
        Variable ArUserIdent
        Variable ArUserInitList_0:
          Variable Execute
          Variable ElementName
          Variable List
        Variable ArUserReleaseRole_0:
          Variable UserName
          Variable RoleName
        Variable ArUserSetPassword_0:
          Variable UserName
          Variable Password
        Variable ArUserSetProperty_0:
          Variable ElementType
          Variable ElementName
          Variable PropertyName
          Variable PropertyValue
        Variable User:
          Variable Command:
            Variable UserCreate
            Variable UserDelete
            Variable UserRename
            Variable PasswordChange
            Variable RoleAssign
            Variable RoleRemove
            Variable Import
            Variable Export
            Variable ListRefresh
            Variable ErrorReset
          Variable Parameter:
            Variable FilePath
            Variable UserName
            Variable UserNameNew
            Variable UserRole
            Variable Password
            Variable PasswordRepeat
            Variable VisuSlotID
          Variable Data:
            Variable Users (EnableArrayElements=True)
            Variable Roles
            Variable Status
            Variable UserActive (EnableArrayElements=True)
          Variable Visualization (EnableArrayElements=True)
          Variable Error:
            Variable No
            Variable State
            Variable Text
      Task ProcessCon:
        Variable AcpAxConfig (EnableArrayElements=True)
          Variable AcpAxConfig[0]:
            Variable MechanicalElements:
              Variable RotaryToLinearTransformation:
                Variable ReferenceDistance (AuditEvents=True, EngineeringUnitId=1)
              Variable Gearbox:
                Variable Input (AuditEvents=True, EURangesId=10)
                Variable Output (AuditEvents=True, EURangesId=10)
            Variable Homing:
              Variable Mode:
                Variable Direct:
                  Variable Position (AuditEvents=True, EngineeringUnitId=1)
          Variable AcpAxConfig[1]:
            Variable Homing:
              Variable Mode:
                Variable Direct:
                  Variable Position (AuditEvents=True, EngineeringUnitId=3)
            Variable MechanicalElements:
              Variable Gearbox:
                Variable Input (AuditEvents=True, EURangesId=10)
                Variable Output (AuditEvents=True, EURangesId=10)
              Variable RotaryToLinearTransformation:
                Variable ReferenceDistance (AuditEvents=True)
        Variable ReadConfig
        Variable WriteConfig
        Variable MC_BR_ProcessConfig_ACP:
          Variable Name
        Variable SelectedAxis
      Task SysServs:
        Variable EthConfig (AutomaticEnable=True)
        Variable ReadEthConfig
        Variable WriteEthConfig
        Variable DTStructureGetTime_0:
          Variable enable
        Variable DTStructureSetTime_0:
          Variable enable
        Variable ClientInfo (EnableArrayElements=True)
        Variable DateTimeCfg (AutomaticEnable=True)
      Task PIDControl:
        Variable MTBasicsPID_0:
          Variable PIDParameters (AutomaticEnable=True)
            Variable IntegrationTime (EngineeringUnitId=12)
            Variable DerivativeTime (EngineeringUnitId=12)
            Variable FilterTime (EngineeringUnitId=12)
          Variable Enable
          Variable MinOut
          Variable MaxOut
          Variable SetValue
          Variable StatusID
        Variable PidControlParameters (AutomaticEnable=True)
          Variable PidParameters:
            Variable IntegrationTime (AuditEvents=True, EURangesId=12, EngineeringUnitId=12)
            Variable DerivativeTime (AuditEvents=True, EURangesId=12, EngineeringUnitId=12)
            Variable FilterTime (AuditEvents=True, EURangesId=12, EngineeringUnitId=12)
            Variable Gain (AuditEvents=True, EURangesId=12)
          Variable MinOut (EURangesId=15)
          Variable MaxOut (EURangesId=16)
        Variable ActValue
        Variable OutValue
        Variable SimulationActive
        Variable MTBasicsOscillationTuning_0:
          Variable Enable
          Variable TuningDone
          Variable TuningActive
        Variable TuningQuality
        Variable PidStatus
      Task IoBrowser:
        Variable TableConfig
        Variable ModuleList (EnableArrayElements=True)
        Variable IoChannel (AutomaticEnable=True)
          Variable IoForcing:
            Variable ForceValue (EURangesId=17, EngineeringUnitId=14)
        Variable IoChannelList (EnableArrayElements=True)
        Variable IoPvList (EnableArrayElements=True)
        Variable SelectedChannel
        Variable SelectedModule
        Variable TableConfigChannels
        Variable IoValueList (EnableArrayElements=True)
        Variable IoChannelTemp:
          Variable IoForcing:
            Variable ForceValue (EURangesId=17, EngineeringUnitId=13)
        Variable StationList (EnableArrayElements=True)
        Variable TableConfigStations
        Variable SelectedStation
        Variable GatIoForcingHandler_0:
          Variable Initializing
      Task CrossCutte
```

### Recipe.uad.bak - 5PPC2200_AL14_000/Connectivity/OpcUA/Recipe.uad.bak
```
OpcUaSource (FileVersion=7, ArVersion=D4.91)
  Aliases:
    ACLAliases:
      ACL (Id=1)
        ACE (RoleName=Service, Access=0x015F)
        ACE (RoleName=Administrators, Access=0x017F)
        ACE (RoleName=Operators, Access=0x015F)
        ACE (RoleName=Everyone, Access=0x015F)
      ACL (Id=3)
        ACE (RoleName=Service, Access=0x01FF)
        ACE (RoleName=Administrators, Access=0x01FF)
        ACE (RoleName=Operators, Access=0x01FF)
        ACE (RoleName=Everyone, Access=0x017F)
    EURangeViolationAliases
    EURangesAliases
    EngineeringUnitAliases
  DefaultView (AclId=3)
    Module <Default>:
      Task Recipe:
        Variable MpRecipeUIConnect:
          Variable Recipe:
            Variable List:
              Variable Names (EnableArrayElements=True)
              Variable SelectedIndex
              Variable LastModified (EnableArrayElements=True)
              Variable PageUp
              Variable PageDown
              Variable RangeStart
              Variable RangeEnd
            Variable Load
            Variable Save
            Variable Delete
            Variable Rename
            Variable NewFileName
            Variable Filter
            Variable Refresh
          Variable New:
            Variable FileName
            Variable Create
          Variable MessageBox:
            Variable Confirm
            Variable Cancel
        Variable HmiRecipe:
          Variable Commands (AutomaticEnable=True)
          Variable Status
          Variable Parameters:
            Variable LastLoadedConfigRecipe
            Variable LastLoadedProductRecipe
            Variable DeviceDataProvider
            Variable DeviceName
            Variable TableConfig
            Variable CategoryDropdown
            Variable EditDialogOpened
            Variable CreateDialogOpened
            Variable ActiveRecipe
        Variable MpRecipeUI_0:
          Variable ErrorReset
          Variable Error
        Variable Parameters (AutomaticEnable=True)
        Variable MachineSettings (AutomaticEnable=True)
        Variable MachineSettingsPreview (AutomaticEnable=True)
        Variable ParametersPreview (AutomaticEnable=True)
        Variable ParametersEdit (AutomaticEnable=True)
        Variable MachineSettingsEdit (AutomaticEnable=True)
        Variable MpRecipe_0:
          Variable ErrorReset
          Variable UpdateNotification
          Variable Error
          Variable Info:
            Variable LastLoadedRecipe
```

### UserX.uad.bak - 5PPC2200_AL14_000/Connectivity/OpcUA/UserX.uad.bak
```
OpcUaSource (FileVersion=7, ArVersion=D4.91)
  Aliases:
    ACLAliases:
      ACL (Id=1)
        ACE (RoleName=Service, Access=0x015F)
        ACE (RoleName=Administrators, Access=0x017F)
        ACE (RoleName=Operators, Access=0x015F)
        ACE (RoleName=Everyone, Access=0x015F)
      ACL (Id=3)
        ACE (RoleName=Service, Access=0x01FF)
        ACE (RoleName=Administrators, Access=0x01FF)
        ACE (RoleName=Operators, Access=0x01FF)
        ACE (RoleName=Everyone, Access=0x017F)
    EURangeViolationAliases
    EURangesAliases
    EngineeringUnitAliases
  DefaultView (AclId=3)
    Module <Default>:
      Task UserX:
        Variable UserXMgrUIConnect (AutomaticEnable=True)
          Variable User:
            Variable List:
              Variable UserNames (EnableArrayElements=True)
              Variable UserOptions (EnableArrayElements=True)
            Variable Info:
              Variable Roles (EnableArrayElements=True)
              Variable AdditionalData (EnableArrayElements=True)
          Variable Import:
            Variable Dialog:
              Variable List:
                Variable FileNames (EnableArrayElements=True)
        Variable MpUserXManagerUI_0:
          Variable ErrorReset
          Variable Error
        Variable UserXLoginUIConnect (AutomaticEnable=True)
        Variable MpUserXLoginUI_0:
          Variable Error
        Variable MpUserXLogin_0:
          Variable Error
```

### UserXMgr.uad.bak - 5PPC2200_AL14_000/Connectivity/OpcUA/UserXMgr.uad.bak
```
OpcUaSource (FileVersion=7, ArVersion=D4.91)
  Aliases:
    ACLAliases:
      ACL (Id=1)
        ACE (RoleName=Service, Access=0x015F)
        ACE (RoleName=Administrators, Access=0x017F)
        ACE (RoleName=Operators, Access=0x015F)
        ACE (RoleName=Everyone, Access=0x015F)
      ACL (Id=3)
        ACE (RoleName=Service, Access=0x01FF)
        ACE (RoleName=Administrators, Access=0x01FF)
        ACE (RoleName=Operators, Access=0x01FF)
        ACE (RoleName=Everyone, Access=0x017F)
    EURangeViolationAliases
    EURangesAliases
    EngineeringUnitAliases
  DefaultView (AclId=3)
    Module <Default>:
      Task UserXMgt:
        Variable UserXMgrUIConnect (AutomaticEnable=True)
          Variable User:
            Variable List:
              Variable UserNames (EnableArrayElements=True)
              Variable UserOptions (EnableArrayElements=True)
            Variable Info:
              Variable Roles (EnableArrayElements=True)
              Variable AdditionalData (EnableArrayElements=True)
          Variable Import:
            Variable Dialog:
              Variable List:
                Variable FileNames (EnableArrayElements=True)
        Variable MpUserXManagerUI_0:
          Variable ErrorReset
          Variable Error
        Variable UserXLoginUIConnect (AutomaticEnable=True)
        Variable MpUserXLoginUI_0:
          Variable Error
        Variable MpUserXLogin_0:
          Variable Error
```

### Cpu.sw.bak - 5PPC2200_AL14_000/Cpu.sw.bak
```
SwConfiguration (CpuAddress=SL1)
  TaskClass Cyclic#1:
    Task MainCtrl (Source=MainControl.MainCtrl.prg, Memory=UserROM, Language=IEC, Debugging=true, Disabled=true)
    Task AxisContro (Source=Infrastructure.AxisTemplate.AxisControl.prg, Memory=UserROM, Language=IEC, Debugging=true, Disabled=true)
    Task AppAxis_1 (Source=MachineControl.AppAxis_1.AppAxis_1.prg, Memory=UserROM, Language=IEC, Debugging=true)
    Task CrossCutte (Source=MachineControl.CrossCutter.CrossCutter.prg, Memory=UserROM, Language=IEC, Debugging=true, Disabled=true)
  TaskClass Cyclic#2:
    Task PIDControl (Source=MainControl.PIDControl.prg, Memory=UserROM, Language=IEC, Debugging=true, Disabled=true)
  TaskClass Cyclic#3
  TaskClass Cyclic#4
  TaskClass Cyclic#5:
    Task UserXMgt (Source=Infrastructure.UserX.UserXMgt.prg, Memory=UserROM, Language=IEC, Debugging=true)
    Task UserMgt (Source=Infrastructure.User.UserMgt.prg, Memory=UserROM, Language=IEC, Debugging=true, Disabled=true)
    Task ProcessCon (Source=Infrastructure.SysServices.ProcessConfig.prg, Memory=UserROM, Language=IEC, Debugging=true, Disabled=true)
    Task AlarmMgr (Source=Infrastructure.AlarmX.AlarmMgr.prg, Memory=UserROM, Language=IEC, Debugging=true)
    Task AuditMgt (Source=Infrastructure.Audit.AuditMgt.prg, Memory=UserROM, Language=IEC, Debugging=true)
    Task DataMgt (Source=Infrastructure.Data.DataMgt.prg, Memory=UserROM, Language=IEC, Debugging=true)
    Task UsbDevLink (Source=Infrastructure.UsbDevLink.UsbDevLink.prg, Memory=UserROM, Language=IEC, Debugging=true)
    Task ReportMgt (Source=Infrastructure.Report.ReportMgt.prg, Memory=UserROM, Language=IEC, Debugging=true)
    Task RecipeMgt (Source=Infrastructure.Recipe.RecipeMgt.prg, Memory=UserROM, Language=IEC, Debugging=true)
    Task BackupMgt (Source=Infrastructure.Backup.BackupMgt.prg, Memory=UserROM, Language=IEC, Debugging=true)
    Task FileMgt (Source=Infrastructure.File.FileMgt.prg, Memory=UserROM, Language=IEC, Debugging=true)
  TaskClass Cyclic#6
  TaskClass Cyclic#7
  TaskClass Cyclic#8:
    Task IoBrowser (Source=Infrastructure.SysServices.IoBrowser.prg, Memory=UserROM, Language=IEC, Debugging=true)
    Task SysServs (Source=Infrastructure.SysServices.SysServs.prg, Memory=UserROM, Language=IEC, Debugging=true)
  DataObjects:
    DataObject McAcpSys (Source=, Memory=UserROM, Language=Binary)
  NcDataObjects:
    NcDataObject McDriveLog (Source=, Memory=UserROM, Language=Binary)
  Binaries:
    BinaryObject McProfGen (Source=, Memory=UserROM, Language=Binary)
    BinaryObject TCData (Source=, Memory=SystemROM, Language=Binary)
    BinaryObject udbdef (Source=, Memory=UserROM, Language=Binary)
    BinaryObject FWRules (Source=, Memory=UserROM, Language=Binary)
    BinaryObject mvLoader (Source=, Memory=UserROM, Language=Binary)
    BinaryObject McAcpSim (Source=, Memory=UserROM, Language=Binary)
    BinaryObject arflatprv (Source=, Memory=UserROM, Language=Binary)
    BinaryObject TCLang (Source=, Memory=UserROM, Language=Binary)
    BinaryObject arcoal (Source=, Memory=UserROM, Language=Binary)
    BinaryObject arsvcreg (Source=, Memory=UserROM, Language=Binary)
    BinaryObject OpcUaSrv (Source=, Memory=UserROM, Language=Binary)
    BinaryObject McAcpDrv (Source=, Memory=UserROM, Language=Binary)
    BinaryObject mCoWebSc (Source=, Memory=UserROM, Language=Binary)
    BinaryObject sysconf (Source=, Memory=SystemROM, Language=Binary)
    BinaryObject Report (Source=, Memory=UserROM, Language=Binary)
    BinaryObject CutterAlm (Source=, Memory=UserROM, Language=Binary)
    BinaryObject Audit (Source=, Memory=UserROM, Language=Binary)
    BinaryObject asfw (Source=, Memory=SystemROM, Language=Binary)
    BinaryObject Data (Source=, Memory=UserROM, Language=Binary)
    BinaryObject UserXlogin (Source=, Memory=UserROM, Language=Binary)
    BinaryObject MachineGrp (Source=, Memory=UserROM, Language=Binary)
    BinaryObject FileMgr (Source=, Memory=UserROM, Language=Binary)
    BinaryObject Role (Source=, Memory=UserROM, Language=Binary)
    BinaryObject User (Source=, Memory=UserROM, Language=Binary)
    BinaryObject Settings (Source=, Memory=UserROM, Language=Binary)
    BinaryObject ashwd (Source=, Memory=SystemROM, Language=Binary)
    BinaryObject ashwac (Source=, Memory=UserROM, Language=Binary)
    BinaryObject CutVirt (Source=, Memory=UserROM, Language=Binary)
    BinaryObject iomap (Source=, Memory=UserROM, Language=Binary)
    BinaryObject arconfig (Source=, Memory=SystemROM, Language=Binary)
    BinaryObject CutAxis (Source=, Memory=UserROM, Language=Binary)
    BinaryObject CutCamAut (Source=, Memory=UserROM, Language=Binary)
    BinaryObject myUnits (Source=, Memory=UserROM, Language=Binary)
    BinaryObject CutterGrp (Source=, Memory=UserROM, Language=Binary)
    BinaryObject Backup (Source=, Memory=UserROM, Language=Binary)
    BinaryObject TC (Source=, Memory=UserROM, Language=Binary)
    BinaryObject BackupFile (Source=, Memory=UserROM, Language=Binary)
    BinaryObject Config (Source=, Memory=UserROM, Language=Binary)
    BinaryObject UserX (Source=, Memory=UserROM, Language=Binary)
    BinaryObject AlarmX (Source=, Memory=UserROM, Language=Binary)
    BinaryObject RecipeXML (Source=, Memory=UserROM, Language=Binary)
    BinaryObject AlarmXHist (Source=, Memory=UserROM, Language=Binary)
    BinaryObject RecipeCSV (Source=, Memory=UserROM, Language=Binary)
    BinaryObject VAppAxis1 (Source=, Memory=UserROM, Language=Binary)
    BinaryObject Axis1Alm (Source=, Memory=UserROM, Language=Binary)
    BinaryObject Axis1Grp (Source=, Memory=UserROM, Language=Binary)
    BinaryObject AppAxis1 (Source=, Memory=UserROM, Language=Binary)
    BinaryObject RecipeFile (Source=, Memory=UserROM, Language=Binary)
    BinaryObject McMechSys (Source=, Memory=UserROM, Language=Binary)
    BinaryObject ConvVirt (Source=, Memory=UserROM, Language=Binary)
    BinaryObject ConvAxis (Source=, Memory=UserROM, Language=Binary)
    BinaryObject ConvGrp (Source=, Memory=UserROM, Language=Binary)
    BinaryObject ConvAlm (Source=, Memory=UserROM, Language=Binary)
    BinaryObject Cutter (Source=, Memory=UserROM, Language=Binary)
    BinaryObject AlmHistory (Source=, Memory=UserROM, Language=Binary)
    BinaryObject Rcp (Source=, Memory=UserROM, Language=Binary)
    BinaryObject Alarm (Source=, Memory=UserROM, Language=Binary)
    BinaryObject UsX (Source=, Memory=UserROM, Language=Binary)
  Libraries:
    LibraryObject operator (Source=Libraries.operator.lby, Memory=UserROM, Language=binary, Debugging=true)
    LibraryObject runtime (Source=Libraries.runtime.lby, Memory=UserROM, Language=binary, Debugging=true)
    LibraryObject astime (Source=Libraries.astime.lby, Memory=UserROM, Language=binary, Debugging=true)
    LibraryObject AsIecCon (Source=Libraries.AsIecCon.lby, Memory=UserROM, Language=binary, Debugging=true)
    LibraryObject brsystem (Source=Libraries.brsystem.lby, Memory=UserROM, Language=binary, Debugging=true)
    LibraryObject sys_lib (Source=Libraries.sys_lib.lby, Memory=UserROM, Language=binary, Debugging=true)
    LibraryObject AsArSdm (Source=Libraries.AsArSdm.lby, Memory=UserROM, Language=binary, Debugging=true)
    LibraryObject FileIO (Source=Libraries.FileIO.lby, Memory=UserROM, Language=binary, Debugging=true)
    LibraryObject standard (Source=Libraries.standard.lby, Memory=UserROM, Language=binary, Debugging=true)
    LibraryObject AsBrStr (Source=Libraries.AsBrStr.lby, Memory=UserROM, Language=binary, Debugging=true)
    LibraryObject asstring (Source=Libraries.asstring.lby, Memory=UserROM, Language=binary, Debugging=true)
    LibraryObject AsBrWStr (Source=Libraries.AsBrWStr.lby, Memory=UserROM, Language=binary, Debugging=true)
    LibraryObject ArUser (Source=Libraries.ArUser.lby, Memory=UserROM, Language=binary, Debugging=true)
    LibraryObject AsMem (Source=Libraries.AsMem.lby, Memory=UserROM, Language=binary, Debugging=true)
    LibraryObject AsARCfg (Source=Libraries.AsARCfg.lby, Memory=UserROM, Language=binary, Debugging=true)
    LibraryObject MTTypes (Source=Libraries.MTTypes.lby, Memory=UserROM, Language=binary, Debugging=true)
    LibraryObject AsZip (Source=Libraries.AsZip.lby, Memory=UserROM, Language=binary, Debugging=true)
    LibraryObject DataObj (Source=Libraries.DataObj.lby, Memory=UserROM, Language=binary, Debugging=true)
    LibraryObject AsUPS (Source=Libraries.AsUPS.lby, Memory=UserROM, Language=binary, Debugging=true)
    LibraryObject AsIO (Source=Libraries.AsIO.lby, Memory=UserROM, Language=binary, Debugging=true)
    LibraryObject AsIOMMan (Source=Libraries.AsIOMMan.lby, Memory=UserROM, Language=binary, Debugging=true)
    LibraryObject Gat (Source=Libraries.Gat.lby, Memory=UserROM, Language=IEC, Debugging=true)
    LibraryObject IoMapMan (Source=Libraries.IoMapMan.lby, Memory=UserROM, Language=Binary, Debugging=true)
    LibraryObject ArCfgMan (Source=Libraries.ArCfgMan.lby, Memory=UserROM, Language=Binary, Debugging=true)
    LibraryObject MTBasics (Source=Libraries.MTBasics.lby, Memory=UserROM, Language=binary, Debugging=true)
    LibraryObject AsUSB (Source=Libraries.AsUSB.lby, Memory=UserROM, Language=binary, Debugging=true)
    LibraryObject CoTrace (Source=Libraries.CoTrace.lby, Memory=UserROM, Language=binary, Debugging=true)
    LibraryObject MpFile (Source=Libraries.MpFile.lby, Memory=UserROM, Language=Binary, Debugging=true)
    LibraryObject MpData (Source=Libraries.MpData.lby, Memory=UserROM, Language=Binary, Debugging=true)
    LibraryObject MpBase (Source=Libraries.MpBase.lby, Memory=UserROM, Language=Binary, Debugging=true)
    LibraryObject MpAxis (Source=Libraries.MpAxis.lby, Memory=UserROM, Language=binary, Debugging=true)
    LibraryObject MpWebXs (Source=Libraries.MpWebXs.lby, Memory=UserROM, Language=Binary, Debugging=true)
    LibraryObject MpAudit (Source=Libraries.MpAudit.lby, Memory=UserROM, Language=Binary, Debugging=true)
    LibraryObject MpRecipe (Source=Libraries.MpRecipe.lby, Memory=UserROM, Language=Binary, Debugging=true)
    LibraryObject MpUserX (Source=Libraries.MpUserX.lby, Memory=UserROM, Language=Binary, Debugging=true)
    LibraryObject MpReport (Source=Libraries.MpReport.lby, Memory=UserROM, Language=Binary, Debugging=true)
    LibraryObject MpAlarmX (Source=Libraries.MpAlarmX.lby, Memory=UserROM, Language=Binary, Debugging=true)
    LibraryObject MpCom (Source=Libraries.MpCom.lby, Memory=UserROM, Language=Binary, Debugging=true)
    LibraryObject MpBackup (Source=Libraries.MpBackup.lby, Memory=UserROM, Language=Binary, Debugging=true)
    LibraryObject McAxis (Source=Libraries.McAxis.lby, Memory=UserROM, Language=binary, Debugging=true)
    LibraryObject McBase (Source=Libraries.McBase.lby, Memory=UserROM, Language=binary, Debugging=true)
    LibraryObject McAcpAx (Source=Libraries.McAcpAx.lby, Memory=UserROM, Language=binary, Debugging=true)
    LibraryObject McPureVAx (Source=Libraries.McPureVAx.lby, Memory=UserROM, Language=binary, Debugging=true)
    LibraryObject McAcpPar (Source=Libraries.McAcpPar.lby, Memory=UserROM, Language=binary, Debugging=true)
    LibraryObject MpServer (Source=Libraries.MpServer.lby, Memory=UserROM, Language=Binary, Debugging=true)
    LibraryObject MpRegMark (Source=Libraries.MpRegMark.lby, Memory=UserROM, Language=Binary, Debugging=true)
    LibraryObject dvframe (Source=Libraries.dvframe.lby, Memory=UserROM, Language=binary, Debugging=true)
    LibraryObject AsIODiag (Source=Libraries.AsIODiag.lby, Memory=UserROM, Language=binary, Debugging=true)
    LibraryObject aseth (Source=, Memory=UserROM, Language=Binary, Debugging=true)
    LibraryObject arssl (Source=, Memory=UserROM, Language=Binary, Debugging=true)
    LibraryObject asepl (Source=, Memory=UserROM, Language=Binary, Debugging=true)
    LibraryObject powerlnk (Source=, Memory=UserROM, Language=Binary, Debugging=true)
    LibraryObject ashw (Source=, Memory=UserROM, Language=Binary, Debugging=true)
    LibraryObject arproject (Source=, Memory=UserROM, Language=Binary, Debugging=true)
    LibraryObject arcert (Source=, Memory=UserROM, Language=Binary, Debugging=true)
    LibraryObject LoggingLib (Source=, Memory=UserROM, Language=Binary, Debugging=true)
    LibraryObject snprintf (Source=, Memory=UserROM, Language=Binary, Debugging=true)
    LibraryObject asarlog (Source=, Memory=UserROM, Language=Binary, Debugging=true)
    LibraryObject asarprof (Source=, Memory=UserROM, Language=Binary, Debugging=true)
```

### TC.textconfig.bak - 5PPC2200_AL14_000/TextSystem/TC.textconfig.bak
```
Element TextConfig (Type=TextConfig)
  Languages:
    UserDefaultLanguage = en
    UserFallbackLanguage = en
    TargetLanguages:
      TargetLanguage[1] = en
      TargetLanguage[2] = zh
      TargetLanguage[3] = de
  TargetFiles:
    TargetFile[1] = mappView.Resources.Texts.HMI_PagesTexts.AxisPageTexts.tmx
    TargetFile[2] = mappView.Resources.Texts.HMI_PagesTexts.ParameterPageTexts.tmx
    TargetFile[3] = mappView.Resources.Texts.HMI_PagesTexts.RecipePageTexts.tmx
    TargetFile[4] = mappView.Resources.Texts.HMI_PagesTexts.AlarmPageTexts.tmx
    TargetFile[5] = mappView.Resources.Texts.HMI_PagesTexts.TrendPageTexts.tmx
    TargetFile[6] = mappView.Resources.Texts.HMI_PagesTexts.HistoryTrendTexts.tmx
    TargetFile[7] = mappView.Resources.Texts.HMI_PagesTexts.ReportPageTexts.tmx
    TargetFile[8] = mappView.Resources.Texts.HMI_PagesTexts.SettingsPageTexts.tmx
    TargetFile[9] = mappView.Resources.Texts.HMI_PagesTexts.UserMgtPageTexts.tmx
    TargetFile[10] = mappView.Resources.Texts.Areas_Texts.TopAreaTexts.tmx
    TargetFile[11] = mappView.Resources.Texts.HMI_PagesTexts.UserManualPageTexts.tmx
    TargetFile[12] = mappView.Resources.Texts.HMI_PagesTexts.WelcomePageTexts.tmx
    TargetFile[13] = mappView.Resources.Texts.Areas_Texts.LoginDialogTexts.tmx
    TargetFile[14] = mappView.Resources.Texts.Areas_Texts.RightNavigationTexts.tmx
    TargetFile[15] = mappView.Resources.Texts.HMI_PagesTexts.DataPageTexts.tmx
    TargetFile[16] = mappView.Resources.Texts.HMI_PagesTexts.DiagnosePageTexts.tmx
    TargetFile[17] = mappView.Resources.Texts.HMI_PagesTexts.AuditPageTexts.tmx
    TargetFile[18] = mappView.Resources.Texts.Infrastructure_Texts.AuditTexts.EventLog.tmx
    TargetFile[19] = mappView.Resources.Texts.Infrastructure_Texts.AuditTexts.UserEvent.tmx
    TargetFile[20] = mappView.Resources.Texts.Infrastructure_Texts.AuditTexts.RecipeEvent.tmx
    TargetFile[21] = mappView.Resources.Texts.Infrastructure_Texts.ToolTipTexts.tmx
    TargetFile[22] = mappView.Resources.Texts.Infrastructure_Texts.CamErrorTexts.tmx
    TargetFile[23] = mappView.Resources.Texts.Areas_Texts.PLCOpenStateTexts.tmx
    TargetFile[24] = mappView.Resources.Texts.Infrastructure_Texts.UserErrorTexts.tmx
    TargetFile[25] = mappView.Resources.Texts.Areas_Texts.PidStateTexts.tmx
    TargetFile[26] = mappView.Resources.Texts.UnitTexts.tmx
    TargetFile[27] = Infrastructure.Recipe.RecipeMgt.RecipeAlarms.tmx
    TargetFile[28] = mappView.Resources.Texts.Infrastructure_Texts.mappAlarms.MpUserXLogin_Alarms.tmx
    TargetFile[29] = mappView.Resources.Texts.Infrastructure_Texts.mappAlarms.MpOeeCore_Alarms.tmx
    TargetFile[30] = mappView.Resources.Texts.Infrastructure_Texts.mappAlarms.MpReportCore_Alarms.tmx
    TargetFile[31] = mappView.Resources.Texts.Infrastructure_Texts.mappAlarms.MpFileManagerUI_Alarms.tmx
    TargetFile[32] = mappView.Resources.Texts.Infrastructure_Texts.mappAlarms.MpMotionAlarms.tmx
    TargetFile[33] = mappView.Resources.Texts.Infrastructure_Texts.AuditTexts.DpDescriptions.tmx
    TargetFile[34] = mappView.Resources.Texts.Infrastructure_Texts.UserList.tmx
    TargetFile[35] = mappView.Resources.Texts.Infrastructure_Texts.IoStationTexts.tmx
    TargetFile[36] = MachineControl.CrossCutter.CrossCutterInfo.tmx
    TargetFile[37] = MachineControl.CrossCutter.CrossCutterAlarms.tmx
    TargetFile[38] = MachineControl.AppAxis_1.AppAxis_1_Info.tmx
    TargetFile[39] = MachineControl.AppAxis_1.AppAxis_1_Alarms.tmx
    TargetFile[40] = Infrastructure.AlarmX.Alarms.tmx
    TargetFile[41] = mappView.Resources.Texts.HMI_PagesTexts.BackupTexts.tmx
    TargetFile[42] = mappView.Resources.Texts.HMI_PagesTexts.FileTexts.tmx
```

### AppAxis1.axis - 5PPC2200_AL14_000/mappMotion/AppAxis_1/AppAxis1.axis
```
Element gMpLinkAppAxis_1 (Type=axis)
  BaseTypeIsReadOnly = 0
  BaseType = Linear
    MeasurementUnit = 5066068
    MeasurementResolutionIsReadOnly = 0
    MeasurementResolution = 0.01
    CountDirectionIsReadOnly = 0
    CountDirection = Standard
  MovementLimitsIsReadOnly = 0
  MovementLimits = Internal
    Position:
      LowerLimitMin = -1.79769313486231E308
      UpperLimitMax = 1.79769313486231E308
      LowerLimit = -1000000000000000000000.0
      UpperLimit = 1000000000000000000000.0
    VelocityIsReadOnly = 0
    Velocity:
      VelocityMax = 3.4E38
      Velocity = 10000
    AccelerationIsReadOnly = 0
    Acceleration:
      AccelerationMax = 3.4E38
      Acceleration = 50000
    DecelerationIsReadOnly = 0
    Deceleration:
      DecelerationMax = 3.4E38
      Deceleration = 50000
  Alarms = MpAlarmX
    mapp.AlarmX.Core.Configuration:
      [0]:
        Message = {$IAT/AppAxis_1/Info/Name} {$Axis/Alarms/System}
        Severity = 20
      [1]:
        Message = {$IAT/AppAxis_1/Info/Name} {$Axis/Alarms/Initialization}
        Severity = 20
      [2]:
        Message = {$IAT/AppAxis_1/Info/Name} {$Axis/Alarms/Parameter}
        Severity = 20
      [3]:
        Message = {$IAT/AppAxis_1/Info/Name} {$Axis/Alarms/Operation}
        Severity = 20
      [4]:
        Message = {$IAT/AppAxis_1/Info/Name} {$Axis/Alarms/DataAccess}
        Severity = 20
      [5]:
        Message = {$IAT/AppAxis_1/Info/Name} {$Axis/Alarms/Syntax}
        Severity = 20
      [9]:
        Message = {$IAT/AppAxis_1/Info/Name} {$Axis/Alarms/Network}
        Severity = 20
      [10]:
        Message = {$IAT/AppAxis_1/Info/Name} {$Axis/Alarms/Encoder}
        Severity = 20
        AdditionalInformation1 = Something wrong with the encoder inside the motor
      [11]:
        Message = {$IAT/AppAxis_1/Info/Name} {$Axis/Alarms/Drive}
        Severity = 20
        AdditionalInformation1 = Acopos Drive Error
      [12]:
        Message = {$IAT/AppAxis_1/Info/Name} {$Axis/Alarms/IO}
        Severity = 20
      [13]:
        Message = {$IAT/AppAxis_1/Info/Name} {$Axis/Alarms/Supply}
        Severity = 20
      [14]:
        Message = {$IAT/AppAxis_1/Info/Name} {$Axis/Alarms/Motor}
        Severity = 20
      [15]:
        Message = {$IAT/AppAxis_1/Info/Name} {$Axis/Alarms/HoldingBrake}
        Severity = 20
```

### VAppAxis1.purevaxcfg - 5PPC2200_AL14_000/mappMotion/AppAxis_1/VAppAxis1.purevaxcfg
```
Element PureVAxCfg_AppAxis_1 (Type=purevaxcfg)
  TypeID = PureVAxConfig
  PureVAxis:
    AxisReference = gAppAxis_1
    Homing:
      Mode = Direct
        Position = 0.0
        ReferencePulse = NotUsed
      RestorePositionVariable
    JerkFilter = NotUsed
```

### Config.mappmotioncfg - 5PPC2200_AL14_000/mappMotion/Config.mappmotioncfg
```
Element MappMotionConfiguration (Type=mappmotioncfg)
  Processing:
    ProcessingTaskClass = 1
  Logger:
    SelectiveLogging = Used
      AdministrativeCommands = Visible
      MovementCommands = Visible
      InformationalCommands = Visible
      SuppressSubcomponents = Inactive
```

### ConvAxis.axis - 5PPC2200_AL14_000/mappMotion/Conveyor/ConvAxis.axis
```
Element gAxisConveyor (Type=axis)
  BaseTypeIsReadOnly = 0
  BaseType = Linear
    MeasurementUnit = 5066068
    MeasurementResolutionIsReadOnly = 0
    MeasurementResolution = 0.01
    CountDirectionIsReadOnly = 0
    CountDirection = Standard
  MovementLimitsIsReadOnly = 0
  MovementLimits = Internal
    Position:
      LowerLimitMin = -1.79769313486231E308
      UpperLimitMax = 1.79769313486231E308
      LowerLimit = -1000000000000000000000.0
      UpperLimit = 1000000000000000000000.0
    VelocityIsReadOnly = 0
    Velocity:
      VelocityMax = 3.4E38
      Velocity = 10000
    AccelerationIsReadOnly = 0
    Acceleration:
      AccelerationMax = 3.4E38
      Acceleration = 50000
    DecelerationIsReadOnly = 0
    Deceleration:
      DecelerationMax = 3.4E38
      Deceleration = 50000
  Alarms = MpAlarmX
    mapp.AlarmX.Core.Configuration:
      [0]:
        Message = {$IAT/Conveyor/Info/Name} {$MpMotion/Alarms/System}
        Severity = 20
      [1]:
        Message = {$IAT/Conveyor/Info/Name} {$MpMotion/Alarms/Initialization}
        Severity = 20
      [2]:
        Message = {$IAT/Conveyor/Info/Name} {$MpMotion/Alarms/Parameter}
        Severity = 20
      [3]:
        Message = {$IAT/Conveyor/Info/Name} {$MpMotion/Alarms/Operation}
        Severity = 20
      [4]:
        Message = {$IAT/Conveyor/Info/Name} {$MpMotion/Alarms/DataAccess}
        Severity = 20
      [5]:
        Message = {$IAT/Conveyor/Info/Name} {$MpMotion/Alarms/Syntax}
        Severity = 20
      [9]:
        Message = {$IAT/Conveyor/Info/Name} {$MpMotion/Alarms/Network}
        Severity = 20
      [10]:
        Message = {$IAT/Conveyor/Info/Name} {$MpMotion/Alarms/Encoder}
        Severity = 20
        AdditionalInformation1 = Something wrong with the encoder inside the motor
      [11]:
        Message = {$IAT/Conveyor/Info/Name} {$MpMotion/Alarms/Drive}
        Severity = 20
        AdditionalInformation1 = Acopos Drive Error
      [12]:
        Message = {$IAT/Conveyor/Info/Name} {$MpMotion/Alarms/IO}
        Severity = 20
      [13]:
        Message = {$IAT/Conveyor/Info/Name} {$MpMotion/Alarms/Supply}
        Severity = 20
      [14]:
        Message = {$IAT/Conveyor/Info/Name} {$MpMotion/Alarms/Motor}
        Severity = 20
      [15]:
        Message = {$IAT/Conveyor/Info/Name} {$MpMotion/Alarms/HoldingBrake}
        Severity = 20
```

### ConvVirt.purevaxcfg - 5PPC2200_AL14_000/mappMotion/Conveyor/ConvVirt.purevaxcfg
```
Element PureVAxCfg_Conveyor (Type=purevaxcfg)
  TypeID = PureVAxConfig
  PureVAxis:
    AxisReference = gAxisConveyor
    Homing:
      Mode = Direct
        Position = 0.0
        ReferencePulse = NotUsed
      RestorePositionVariable
    JerkFilter = NotUsed
```

### CutAxis.axis - 5PPC2200_AL14_000/mappMotion/CrossCutter/CutAxis.axis
```
Element gAxisCrossCutter (Type=axis)
  BaseTypeIsReadOnly = 0
  BaseType = RotaryPeriodic
    MeasurementUnitIsReadOnly = 0
    MeasurementUnit = 17476
    MeasurementResolutionIsReadOnly = 0
    MeasurementResolution = 0.01
    CountDirectionIsReadOnly = 0
    CountDirection = Inverse
    PeriodSettings:
      Period = 360
  MovementLimitsIsReadOnly = 0
  MovementLimits = Internal
    Position:
      LowerLimitMin = -1.79769313486231E308
      UpperLimitMax = 1.79769313486231E308
      LowerLimit = -1000.0
      UpperLimit = 1000.0
    VelocityIsReadOnly = 0
    Velocity:
      VelocityMax = 3.4E38
      Velocity = 500000
    AccelerationIsReadOnly = 0
    Acceleration:
      AccelerationMax = 3.4E38
      Acceleration = 5000000
    DecelerationIsReadOnly = 0
    Deceleration:
      DecelerationMax = 3.4E38
      Deceleration = 5000000
  Alarms = MpAlarmX
    mapp.AlarmX.Core.Configuration:
      [0]:
        Message = {$CrossCutter/Info/Name} : {$Axis/Alarms/System}
        Severity = 20
      [1]:
        Message = {$CrossCutter/Info/Name} : {$Axis/Alarms/Initialization}
        Severity = 20
      [2]:
        Message = {$CrossCutter/Info/Name} : {$Axis/Alarms/Parameter}
        Severity = 20
      [3]:
        Message = {$CrossCutter/Info/Name} : {$Axis/Alarms/Operation}
        Severity = 20
      [4]:
        Message = {$CrossCutter/Info/Name} : {$Axis/Alarms/DataAccess}
        Severity = 20
      [5]:
        Message = {$CrossCutter/Info/Name} : {$Axis/Alarms/Syntax}
        Severity = 20
      [9]:
        Message = {$CrossCutter/Info/Name} : {$Axis/Alarms/Network}
        Severity = 20
      [10]:
        Message = {$CrossCutter/Info/Name} : {$Axis/Alarms/Encoder}
        Severity = 20
      [11]:
        Message = {$Axis/Alarms/Drive}
        Severity = 20
      [12]:
        Message = {$Axis/Alarms/IO}
        Severity = 20
      [13]:
        Message = {$Axis/Alarms/Supply}
        Severity = 20
      [14]:
        Message = {$Axis/Alarms/Motor}
        Severity = 20
      [15]:
        Message = {$Axis/Alarms/HoldingBrake}
        Severity = 20
```
